  MoveL 1334 to (137.98, -40.97, -45.71) mm, rotated rx -73.13 ry 0 rz 74.07 deg; joints [-2.429, -86.299, 124.187, -182.116, 24.075, 198.51, -176.517]
  MoveL 1335 to (137.95, -41.43, -45.38) mm, rotated rx -73.26 ry 0 rz 73.89 deg; joints [-2.385, -86.31, 124.184, -182.011, 24.075, 198.293, -176.321]
  MoveL 1336 to (137.95, -41.9, -44.95) mm, rotated rx -73.26 ry 0 rz 73.89 deg; joints [-2.363, -86.282, 124.153, -181.958, 24.075, 198.25, -176.318]
  MoveL 1337 to (138.12, -44.92, -41.35) mm, rotated rx -75.02 ry 0 rz 72.24 deg; joints [-1.813, -86.514, 124.201, -180.651, 24.074, 195.429, -174.469]
  MoveL 1338 to (137.32, -48.01, -40.54) mm, rotated rx -75.35 ry 0 rz 70.98 deg; joints [-1.704, -86.538, 124.192, -180.391, 24.074, 194.895, -173.18]
  MoveL 1339 to (137.34, -47.93, -40.55) mm, rotated rx -75.14 ry 0 rz 70.12 deg; joints [-1.748, -86.7, 124.344, -180.494, 24.074, 195.181, -172.312]
  MoveL 1340 to (135.25, -51.11, -43.62) mm, rotated rx -73.93 ry 0 rz 68.65 deg; joints [-2.159, -86.606, 124.375, -181.473, 24.074, 197.191, -170.974]
  MoveL 1341 to (134.45, -52.71, -44.19) mm, rotated rx -73.93 ry 0 rz 68.65 deg; joints [-2.187, -86.465, 124.261, -181.539, 24.075, 197.244, -171.001]
  MoveL 1342 to (134.28, -53.17, -44.17) mm, rotated rx -73.94 ry 0 rz 68.46 deg; joints [-2.183, -86.466, 124.261, -181.53, 24.075, 197.226, -170.805]
  MoveL 1343 to (133.34, -55.46, -44.11) mm, rotated rx -73.97 ry 0 rz 67.44 deg; joints [-2.175, -86.474, 124.266, -181.512, 24.074, 197.187, -169.78]
  MoveL 1344 to (132.43, -57.68, -44.06) mm, rotated rx -73.98 ry 0 rz 66.48 deg; joints [-2.169, -86.476, 124.265, -181.497, 24.074, 197.156, -168.826]
  MoveL 1345 to (132.15, -58.44, -43.91) mm, rotated rx -73.98 ry 0 rz 66.48 deg; joints [-2.161, -86.417, 124.212, -181.478, 24.074, 197.14, -168.832]
  MoveL 1346 to (131.99, -58.95, -43.73) mm, rotated rx -74.06 ry 0 rz 66.28 deg; joints [-2.136, -86.423, 124.21, -181.419, 24.074, 197.018, -168.614]
  MoveL 1347 to (131, -62.6, -41.54) mm, rotated rx -74.84 ry 0 rz 64.98 deg; joints [-1.862, -86.452, 124.16, -180.765, 24.074, 195.708, -167.238]
  MoveL 1348 to (128.38, -67.77, -41.64) mm, rotated rx -74.94 ry 0 rz 62.15 deg; joints [-1.845, -86.56, 124.248, -180.727, 24.074, 195.572, -164.387]
  MoveL 1349 to (145.45, -76.79, -46.84) mm, rotated rx -74.94 ry 0 rz 62.15 deg; joints [-2.108, -87.321, 123.937, -181.362, 24.074, 196.101, -163.319]
  Set speed (1000.0 mm/s)
  MoveL 1350 to (145.71, -79, -42.14) mm, rotated rx -75.13 ry 0 rz 62.13 deg; joints [-1.831, -87.249, 123.803, -180.699, 24.074, 195.37, -163.234]
  Set speed (5.0 mm/s)
  MoveL 1351 to (128.62, -69.96, -37.01) mm, rotated rx -75.13 ry 0 rz 62.13 deg; joints [-1.573, -86.483, 124.11, -180.078, 24.074, 194.858, -164.306]
  Set speed (16.7 mm/s)
  MoveL 1352 to (129.85, -68.52, -35.3) mm, rotated rx -75.8 ry 0 rz 62.86 deg; joints [-1.345, -86.527, 124.09, -179.536, 24.074, 193.748, -164.966]
  MoveL 1353 to (129.85, -68.52, -35.32) mm, rotated rx -76.99 ry 0 rz 63 deg; joints [-1.094, -86.543, 124.043, -178.936, 24.074, 192.069, -165.05]
  MoveL 1354 to (129.74, -69.29, -34.22) mm, rotated rx -77.8 ry 0 rz 62.22 deg; joints [-0.864, -86.677, 124.104, -178.388, 24.074, 190.808, -164.197]
  MoveL 1355 to (129.04, -70.88, -33.63) mm, rotated rx -78.03 ry 0 rz 61.54 deg; joints [-0.785, -86.689, 124.097, -178.199, 24.074, 190.424, -163.504]
  MoveL 1356 to (128.8, -71.45, -33.34) mm, rotated rx -78.08 ry 0 rz 61.44 deg; joints [-0.759, -86.666, 124.071, -178.138, 24.074, 190.321, -163.401]
  MoveL 1357 to (128.09, -73.34, -31.98) mm, rotated rx -78.67 ry 0 rz 60.52 deg; joints [-0.565, -86.719, 124.074, -177.674, 24.074, 189.356, -162.441]
  MoveL 1358 to (127.59, -74.37, -31.59) mm, rotated rx -78.82 ry 0 rz 60.08 deg; joints [-0.513, -86.726, 124.068, -177.549, 24.074, 189.101, -161.985]
  MoveL 1359 to (123.08, -82.67, -28.71) mm, rotated rx -79.95 ry 0 rz 56.4 deg; joints [-0.125, -86.775, 124.03, -176.622, 24.074, 187.214, -158.23]
  MoveL 1360 to (139.48, -93.57, -32.2) mm, rotated rx -79.95 ry 0 rz 56.4 deg; joints [-0.294, -87.571, 123.736, -177.018, 24.074, 187.514, -157.133]
  Set speed (1000.0 mm/s)
  MoveL 1361 to (86.56, -126.27, -76.23) mm, rotated rx -62.7 ry 0 rz 34.53 deg; joints [-6.054, -85.789, 124.002, -190.764, 24.074, 215.943, -137.619]
  Set speed (5.0 mm/s)
  MoveL 1362 to (76.48, -111.63, -67.06) mm, rotated rx -62.7 ry 0 rz 34.53 deg; joints [-5.589, -85.188, 124.406, -189.599, 24.074, 214.927, -138.553]
  Set speed (16.7 mm/s)
  MoveL 1363 to (78.17, -110.46, -67.04) mm, rotated rx -62.7 ry 0 rz 35.27 deg; joints [-5.589, -85.211, 124.425, -189.599, 24.074, 214.927, -139.295]
  MoveL 1364 to (82.31, -108.27, -65.64) mm, rotated rx -63.33 ry 0 rz 37.57 deg; joints [-5.395, -85.243, 124.366, -189.141, 24.074, 213.928, -141.481]
  MoveL 1365 to (83.1, -107.77, -65.47) mm, rotated rx -63.37 ry 0 rz 37.82 deg; joints [-5.379, -85.267, 124.367, -189.118, 24.033, 213.874, -141.742]
  MoveL 1366 to (86.56, -105.46, -64.75) mm, rotated rx -63.68 ry 0 rz 39.58 deg; joints [-5.284, -85.309, 124.362, -188.893, 24.033, 213.389, -143.445]
  MoveL 1367 to (90.08, -104.34, -61.68) mm, rotated rx -65.21 ry 0 rz 41.53 deg; joints [-4.83, -85.421, 124.266, -187.819, 24.033, 211.007, -145.135]
  MoveL 1368 to (92.29, -104.07, -58.82) mm, rotated rx -66.58 ry 0 rz 42.45 deg; joints [-4.417, -85.567, 124.225, -186.84, 24.033, 208.859, -145.827]
  MoveL 1369 to (93.65, -103.42, -57.81) mm, rotated rx -66.58 ry 0 rz 42.45 deg; joints [-4.368, -85.649, 124.225, -186.766, 23.858, 208.808, -145.916]
  MoveL 1370 to (94.29, -102.92, -57.66) mm, rotated rx -66.61 ry 0 rz 42.54 deg; joints [-4.357, -85.68, 124.226, -186.757, 23.785, 208.78, -146.046]
  MoveL 1371 to (95.59, -101.74, -57.6) mm, rotated rx -66.63 ry 0 rz 43.26 deg; joints [-4.348, -85.683, 124.225, -186.737, 23.786, 208.737, -146.762]
  MoveL 1372 to (97.07, -100.77, -56.82) mm, rotated rx -67.03 ry 0 rz 44.34 deg; joints [-4.227, -85.661, 124.161, -186.448, 23.786, 208.107, -147.797]
  MoveL 1373 to (99.36, -99.94, -54.29) mm, rotated rx -68.34 ry 0 rz 45.63 deg; joints [-3.838, -85.738, 124.083, -185.516, 23.786, 206.052, -148.895]
  MoveL 1374 to (99.89, -99.67, -53.81) mm, rotated rx -68.34 ry 0 rz 45.63 deg; joints [-3.814, -85.771, 124.083, -185.472, 23.718, 206.019, -148.928]
  MoveL 1375 to (100.33, -99.39, -53.5) mm, rotated rx -68.42 ry 0 rz 45.75 deg; joints [-3.784, -85.792, 124.084, -185.404, 23.696, 205.89, -149.049]
  MoveL 1376 to (103.28, -97.29, -51.72) mm, rotated rx -69.14 ry 0 rz 47.19 deg; joints [-3.549, -85.876, 124.073, -184.84, 23.696, 204.714, -150.376]
  MoveL 1377 to (103.68, -96.97, -51.52) mm, rotated rx -69.17 ry 0 rz 47.28 deg; joints [-3.533, -85.894, 124.073, -184.805, 23.665, 204.653, -150.482]
  MoveL 1378 to (105.78, -94.99, -50.95) mm, rotated rx -69.35 ry 0 rz 48.27 deg; joints [-3.468, -85.936, 124.074, -184.658, 23.62, 204.355, -151.47]
  MoveL 1379 to (106.4, -94.3, -50.95) mm, rotated rx -69.35 ry 0 rz 48.27 deg; joints [-3.469, -86.006, 124.135, -184.661, 23.62, 204.358, -151.46]
  MoveL 1380 to (106.81, -93.76, -51.06) mm, rotated rx -69.31 ry 0 rz 48.54 deg; joints [-3.485, -86.001, 124.136, -184.698, 23.62, 204.434, -151.739]
  MoveL 1381 to (109.17, -90.01, -52.73) mm, rotated rx -68.69 ry 0 rz 50.1 deg; joints [-3.694, -85.967, 124.18, -185.203, 23.618, 205.459, -153.389]
  MoveL 1382 to (109.1, -90.07, -52.8) mm, rotated rx -68.9 ry 0 rz 51.22 deg; joints [-3.648, -85.766, 123.992, -185.092, 23.618, 205.151, -154.518]
  MoveL 1383 to (110.45, -89.31, -51.3) mm, rotated rx -69.51 ry 0 rz 51.79 deg; joints [-3.451, -85.835, 123.982, -184.615, 23.618, 204.161, -155.002]
  MoveL 1384 to (110.71, -89.18, -50.98) mm, rotated rx -69.68 ry 0 rz 51.94 deg; joints [-3.4, -85.846, 123.974, -184.494, 23.618, 203.894, -155.123]
  MoveL 1385 to (114.23, -86.61, -47.5) mm, rotated rx -70.95 ry 0 rz 53.48 deg; joints [-2.968, -86.008, 123.97, -183.452, 23.618, 201.783, -156.483]
  MoveL 1386 to (115.16, -85.68, -46.95) mm, rotated rx -70.95 ry 0 rz 53.48 deg; joints [-2.942, -86.105, 124.036, -183.392, 23.585, 201.736, -156.483]
  MoveL 1387 to (115.49, -85.28, -46.88) mm, rotated rx -70.98 ry 0 rz 53.69 deg; joints [-2.933, -86.108, 124.036, -183.371, 23.585, 201.692, -156.687]
  MoveL 1388 to (116.72, -83.72, -46.58) mm, rotated rx -71.09 ry 0 rz 54.5 deg; joints [-2.893, -86.116, 124.03, -183.275, 23.585, 201.495, -157.483]
  MoveL 1389 to (117.65, -83.33, -44.95) mm, rotated rx -71.52 ry 0 rz 54.9 deg; joints [-2.724, -86.154, 124.01, -182.866, 23.585, 200.738, -157.816]
  MoveL 1390 to (118.89, -81.86, -44.41) mm, rotated rx -71.96 ry 0 rz 55.31 deg; joints [-2.606, -86.254, 124.06, -182.581, 23.585, 200.066, -158.172]
  MoveL 1391 to (119.23, -81.32, -44.49) mm, rotated rx -71.93 ry 0 rz 55.56 deg; joints [-2.618, -86.251, 124.061, -182.609, 23.585, 200.122, -158.429]
  MoveL 1392 to (122.81, -74.48, -46.64) mm, rotated rx -71.1 ry 0 rz 58.48 deg; joints [-2.897, -86.199, 124.103, -183.283, 23.585, 201.496, -161.446]
  MoveL 1393 to (123.08, -74.04, -46.65) mm, rotated rx -71.07 ry 0 rz 58.84 deg; joints [-2.904, -86.181, 124.102, -183.295, 23.632, 201.537, -161.778]
  MoveL 1394 to (125.13, -70.14, -47.21) mm, rotated rx -70.84 ry 0 rz 60.59 deg; joints [-2.978, -86.159, 124.107, -183.474, 23.632, 201.908, -163.564]
  MoveL 1395 to (125.67, -68.6, -48.04) mm, rotated rx -70.81 ry 0 rz 60.59 deg; joints [-3.029, -86.265, 124.215, -183.596, 23.632, 202.041, -163.568]
  MoveL 1396 to (125.64, -67.91, -49.09) mm, rotated rx -70.78 ry 0 rz 60.59 deg; joints [-3.087, -86.292, 124.256, -183.737, 23.632, 202.179, -163.586]
  MoveL 1397 to (124.81, -67.96, -51.11) mm, rotated rx -70.74 ry 0 rz 60.59 deg; joints [-3.197, -86.235, 124.256, -183.996, 23.676, 202.429, -163.605]
  MoveL 1398 to (123.74, -68.7, -52.68) mm, rotated rx -69.66 ry 0 rz 59.95 deg; joints [-3.498, -86.168, 124.3, -184.721, 23.677, 204.099, -163.092]
  MoveL 1399 to (123.37, -68.58, -53.7) mm, rotated rx -69.24 ry 0 rz 59.92 deg; joints [-3.633, -86.121, 124.306, -185.046, 23.677, 204.775, -163.118]
  MoveL 1400 to (122.17, -69.3, -55.43) mm, rotated rx -67.67 ry 0 rz 59.88 deg; joints [-4.037, -85.916, 124.306, -185.994, 23.78, 207.108, -163.209]
  MoveL 1401 to (122.63, -67.73, -56.41) mm, rotated rx -67.27 ry 0 rz 60.52 deg; joints [-4.165, -85.868, 124.311, -186.3, 23.78, 207.748, -163.921]
  MoveL 1402 to (123.25, -65.21, -58) mm, rotated rx -66.64 ry 0 rz 61.52 deg; joints [-4.371, -85.791, 124.324, -186.793, 23.78, 208.777, -165.028]
  MoveL 1403 to (123.68, -64.08, -58.35) mm, rotated rx -66.37 ry 0 rz 62.29 deg; joints [-4.441, -85.732, 124.324, -186.941, 23.857, 209.16, -165.779]
  MoveL 1404 to (123.84, -63.54, -58.59) mm, rotated rx -66.37 ry 0 rz 62.29 deg; joints [-4.455, -85.77, 124.361, -186.974, 23.857, 209.187, -165.78]
  MoveL 1405 to (124.29, -61.65, -59.63) mm, rotated rx -65.93 ry 0 rz 63.09 deg; joints [-4.593, -85.707, 124.362, -187.304, 23.857, 209.892, -166.655]
  MoveL 1406 to (124.3, -61.62, -59.61) mm, rotated rx -66.05 ry 0 rz 64.34 deg; joints [-4.56, -85.492, 124.167, -187.224, 23.857, 209.703, -167.922]
  MoveL 1407 to (126.02, -59.94, -57.71) mm, rotated rx -66.83 ry 0 rz 65.26 deg; joints [-4.311, -85.596, 124.158, -186.63, 23.857, 208.448, -168.706]
  MoveL 1408 to (128.44, -59.64, -52.46) mm, rotated rx -69.46 ry 0 rz 66.08 deg; joints [-3.521, -85.835, 124.075, -184.743, 23.857, 204.31, -169.145]
  MoveL 1409 to (128.8, -59.51, -51.74) mm, rotated rx -69.54 ry 0 rz 66.1 deg; joints [-3.469, -85.868, 124.085, -184.62, 23.857, 204.13, -169.145]
  MoveL 1410 to (129.78, -58.91, -49.96) mm, rotated rx -70.26 ry 0 rz 66.48 deg; joints [-3.233, -85.946, 124.072, -184.057, 23.855, 202.958, -169.423]
  MoveL 1411 to (130.23, -58.65, -49.07) mm, rotated rx -70.48 ry 0 rz 66.57 deg; joints [-3.143, -85.991, 124.081, -183.841, 23.855, 202.559, -169.462]
  MoveL 1412 to (132.89, -56.13, -44.69) mm, rotated rx -72.23 ry 0 rz 67.91 deg; joints [-2.565, -86.163, 124.047, -182.456, 23.855, 199.694, -170.572]
  MoveL 1413 to (133.87, -54.54, -43.72) mm, rotated rx -72.23 ry 0 rz 67.91 deg; joints [-2.517, -86.301, 124.138, -182.348, 23.806, 199.607, -170.572]
  MoveL 1414 to (134.4, -52.63, -44.42) mm, rotated rx -72.23 ry 0 rz 67.91 deg; joints [-2.555, -86.439, 124.266, -182.438, 23.802, 199.68, -170.568]
  MoveL 1415 to (134.45, -52.04, -44.98) mm, rotated rx -72.01 ry 0 rz 68.13 deg; joints [-2.628, -86.418, 124.271, -182.615, 23.802, 200.044, -170.823]
  MoveL 1416 to (134.35, -51.3, -46.09) mm, rotated rx -72.01 ry 0 rz 68.13 deg; joints [-2.685, -86.451, 124.317, -182.75, 23.802, 200.154, -170.838]
  MoveL 1417 to (132.92, -49.01, -52.29) mm, rotated rx -68.94 ry 0 rz 69.21 deg; joints [-3.624, -86.082, 124.317, -184.994, 23.838, 205.029, -172.299]
  MoveL 1418 to (133.31, -45.82, -54.18) mm, rotated rx -68.18 ry 0 rz 70.48 deg; joints [-3.873, -85.993, 124.328, -185.589, 23.838, 206.272, -173.685]
  MoveL 1419 to (133.02, -44.52, -55.95) mm, rotated rx -68.18 ry 0 rz 70.48 deg; joints [-3.963, -86.046, 124.406, -185.806, 23.838, 206.446, -173.717]
  MoveL 1420 to (132.73, -44.42, -56.71) mm, rotated rx -68.1 ry 0 rz 70.49 deg; joints [-4.017, -86.023, 124.406, -185.936, 23.838, 206.629, -173.751]
  MoveL 1421 to (132.12, -44.47, -58.08) mm, rotated rx -67.54 ry 0 rz 70.38 deg; joints [-4.198, -85.953, 124.414, -186.368, 23.838, 207.536, -173.74]
  MoveL 1422 to (131.58, -43.17, -60.26) mm, rotated rx -66.1 ry 0 rz 70.89 deg; joints [-4.592, -85.779, 124.417, -187.308, 23.838, 209.722, -174.459]
  MoveL 1423 to (131.38, -42.9, -60.88) mm, rotated rx -66.1 ry 0 rz 70.89 deg; joints [-4.624, -85.78, 124.431, -187.384, 23.838, 209.782, -174.474]
  MoveL 1424 to (131.19, -42.76, -61.38) mm, rotated rx -65.89 ry 0 rz 70.92 deg; joints [-4.69, -85.752, 124.433, -187.542, 23.838, 210.117, -174.541]
  MoveL 1425 to (130.01, -41.88, -64.4) mm, rotated rx -64.63 ry 0 rz 71.11 deg; joints [-5.089, -85.574, 124.446, -188.493, 23.838, 212.139, -174.964]
  MoveL 1426 to (130.03, -41.89, -64.35) mm, rotated rx -63.97 ry 0 rz 71.59 deg; joints [-5.213, -85.465, 124.446, -188.743, 23.975, 212.984, -175.43]
  MoveL 1427 to (130.19, -37.44, -66.76) mm, rotated rx -62.96 ry 0 rz 73.39 deg; joints [-5.527, -85.314, 124.456, -189.488, 23.975, 214.583, -177.435]
  MoveL 1428 to (129.62, -36.05, -68.6) mm, rotated rx -62.96 ry 0 rz 73.39 deg; joints [-5.622, -85.357, 124.534, -189.714, 23.975, 214.762, -177.483]
  MoveL 1429 to (129.03, -35.2, -70.14) mm, rotated rx -62.01 ry 0 rz 73.73 deg; joints [-5.88, -85.215, 124.534, -190.323, 23.978, 216.195, -177.992]
  MoveL 1430 to (128.75, -34.95, -70.79) mm, rotated rx -61.95 ry 0 rz 73.75 deg; joints [-5.923, -85.204, 124.543, -190.423, 23.978, 216.325, -178.035]
  MoveL 1431 to (128.62, -34.84, -71.06) mm, rotated rx -61.16 ry 0 rz 74.22 deg; joints [-6.085, -85.07, 124.543, -190.76, 24.099, 217.374, -178.54]
  MoveL 1432 to (128.52, -33.37, -71.94) mm, rotated rx -60.78 ry 0 rz 74.81 deg; joints [-6.199, -85.009, 124.547, -191.029, 24.099, 217.961, -179.22]
  MoveL 1433 to (128.3, -32.51, -72.73) mm, rotated rx -60.78 ry 0 rz 74.81 deg; joints [-6.241, -85.045, 124.597, -191.128, 24.099, 218.039, -179.24]
  MoveL 1434 to (128.05, -32.17, -73.32) mm, rotated rx -60.73 ry 0 rz 74.84 deg; joints [-6.28, -85.039, 124.611, -191.219, 24.099, 218.159, -179.294]
  MoveL 1435 to (127.47, -31.67, -74.53) mm, rotated rx -60.2 ry 0 rz 74.99 deg; joints [-6.438, -84.951, 124.616, -191.591, 24.099, 218.974, -179.554]
  MoveL 1436 to (126.85, -29.7, -76.38) mm, rotated rx -59.02 ry 0 rz 75.96 deg; joints [-6.771, -84.988, 125.113, -191.94, 25.126, 220.344, -180]
  MoveL 1437 to (126.72, -29.34, -76.74) mm, rotated rx -58.91 ry 0 rz 76.06 deg; joints [-6.814, -85.013, 125.204, -191.969, 25.294, 220.465, -180]
  MoveL 1438 to (125.84, -27.3, -78.9) mm, rotated rx -57.96 ry 0 rz 76.84 deg; joints [-7.131, -85.152, 125.88, -192.137, 26.641, 221.44, -180]
  MoveL 1439 to (125.36, -26.75, -79.85) mm, rotated rx -57.96 ry 0 rz 76.84 deg; joints [-7.181, -85.165, 125.931, -192.227, 26.686, 221.505, -180]
  MoveL 1440 to (124.53, -26.64, -81.17) mm, rotated rx -57.8 ry 0 rz 76.87 deg; joints [-7.277, -85.126, 125.99, -192.382, 26.821, 221.763, -180]
  MoveL 1441 to (122.66, -27.32, -83.76) mm, rotated rx -56.63 ry 0 rz 76.37 deg; joints [-7.618, -84.902, 125.994, -193.109, 26.821, 223.479, -179.787]
  MoveL 1442 to (120.31, -27.21, -87.13) mm, rotated rx -54.87 ry 0 rz 76.1 deg; joints [-8.096, -84.582, 126.011, -194.127, 26.821, 225.985, -179.937]
  MoveL 1443 to (119.84, -27.31, -87.74) mm, rotated rx -54.87 ry 0 rz 76.1 deg; joints [-8.125, -84.551, 126.011, -194.178, 26.848, 226.019, -179.947]
  MoveL 1444 to (119.51, -27.47, -88.15) mm, rotated rx -54.68 ry 0 rz 75.99 deg; joints [-8.179, -84.513, 126.012, -194.292, 26.848, 226.294, -179.886]
  MoveL 1445 to (115.59, -30.1, -92.42) mm, rotated rx -52.79 ry 0 rz 74.41 deg; joints [-8.711, -84.104, 126.015, -195.418, 26.848, 228.993, -178.81]
  MoveL 1446 to (115.26, -30.28, -92.76) mm, rotated rx -52.59 ry 0 rz 74.25 deg; joints [-8.762, -84.07, 126.021, -195.526, 26.848, 229.272, -178.705]
  MoveL 1447 to (111.45, -33.08, -96.4) mm, rotated rx -50.93 ry 0 rz 72.51 deg; joints [-9.215, -83.699, 126.028, -196.481, 26.848, 231.613, -177.43]
  MoveL 1448 to (110.88, -33.62, -96.87) mm, rotated rx -50.85 ry 0 rz 72.38 deg; joints [-9.25, -83.65, 126.028, -196.526, 26.9, 231.715, -177.302]
  MoveL 1449 to (109.03, -35.76, -98.19) mm, rotated rx -50.24 ry 0 rz 71.16 deg; joints [-9.414, -83.504, 126.028, -196.869, 26.901, 232.572, -176.255]
  MoveL 1450 to (105.97, -37.85, -100.72) mm, rotated rx -48.8 ry 0 rz 69.4 deg; joints [-9.771, -83.244, 126.083, -197.617, 26.901, 234.531, -174.884]
  MoveL 1451 to (105.56, -38.13, -101.04) mm, rotated rx -48.65 ry 0 rz 69.21 deg; joints [-9.81, -83.208, 126.083, -197.698, 26.901, 234.736, -174.743]
  MoveL 1452 to (102.4, -40.39, -103.39) mm, rotated rx -47.47 ry 0 rz 67.57 deg; joints [-10.109, -82.943, 126.104, -198.318, 26.901, 236.342, -173.448]
  MoveL 1453 to (101.99, -40.57, -103.73) mm, rotated rx -47.27 ry 0 rz 67.37 deg; joints [-10.157, -82.905, 126.112, -198.417, 26.901, 236.61, -173.305]
  MoveL 1454 to (97.91, -42.95, -106.66) mm, rotated rx -45.71 ry 0 rz 65.33 deg; joints [-10.536, -82.565, 126.153, -199.2, 26.901, 238.696, -171.734]
  MoveL 1455 to (96.76, -44.15, -107.22) mm, rotated rx -45.71 ry 0 rz 65.33 deg; joints [-10.552, -82.429, 126.069, -199.214, 26.926, 238.696, -171.762]
  MoveL 1456 to (95.06, -46.9, -107.57) mm, rotated rx -45.52 ry 0 rz 63.53 deg; joints [-10.599, -82.396, 126.083, -199.311, 26.926, 238.956, -170.017]
  MoveL 1457 to (92.2, -49.19, -109.03) mm, rotated rx -44.59 ry 0 rz 61.21 deg; joints [-10.814, -82.269, 126.168, -199.753, 26.926, 240.175, -167.952]
  MoveL 1458 to (91.24, -50.42, -109.28) mm, rotated rx -44.59 ry 0 rz 61.21 deg; joints [-10.814, -82.145, 126.073, -199.749, 26.927, 240.167, -167.981]
  MoveL 1459 to (90.83, -51.64, -109.04) mm, rotated rx -44.6 ry 0 rz 61.05 deg; joints [-10.793, -82.085, 126.01, -199.705, 26.927, 240.124, -167.816]
  MoveL 1460 to (90.6, -53.29, -108.43) mm, rotated rx -44.94 ry 0 rz 60.2 deg; joints [-10.715, -82.159, 126, -199.544, 26.928, 239.685, -166.862]
  MoveL 1461 to (90.59, -53.38, -108.39) mm, rotated rx -45.04 ry 0 rz 59.12 deg; joints [-10.712, -82.315, 126.115, -199.544, 26.925, 239.586, -165.746]
  MoveL 1462 to (89.12, -54.97, -108.83) mm, rotated rx -44.81 ry 0 rz 57.95 deg; joints [-10.768, -82.263, 126.123, -199.658, 26.925, 239.897, -164.653]
  MoveL 1463 to (88.6, -55.68, -108.89) mm, rotated rx -44.81 ry 0 rz 57.95 deg; joints [-10.764, -82.196, 126.069, -199.649, 26.925, 239.888, -164.665]
  MoveL 1464 to (88.21, -56.59, -108.74) mm, rotated rx -44.81 ry 0 rz 57.86 deg; joints [-10.749, -82.144, 126.017, -199.617, 26.925, 239.86, -164.569]
  MoveL 1465 to (87.77, -58.17, -108.26) mm, rotated rx -45.07 ry 0 rz 57.01 deg; joints [-10.688, -82.202, 126.008, -199.491, 26.925, 239.515, -163.635]
  MoveL 1466 to (87.47, -59.22, -107.93) mm, rotated rx -45.14 ry 0 rz 56.72 deg; joints [-10.658, -82.188, 125.973, -199.429, 26.925, 239.406, -163.314]
  MoveL 1467 to (87.01, -63.11, -106.08) mm, rotated rx -46.14 ry 0 rz 54.84 deg; joints [-10.419, -82.41, 125.945, -198.939, 26.925, 238.081, -161.137]
  MoveL 1468 to (87.5, -64.69, -104.72) mm, rotated rx -46.14 ry 0 rz 54.84 deg; joints [-10.346, -82.395, 125.874, -198.786, 26.925, 237.975, -161.064]
  MoveL 1469 to (88.16, -65.07, -103.92) mm, rotated rx -46.27 ry 0 rz 54.83 deg; joints [-10.288, -82.454, 125.873, -198.668, 26.925, 237.766, -160.984]
  MoveL 1470 to (89.29, -65.35, -102.77) mm, rotated rx -46.86 ry 0 rz 55.05 deg; joints [-10.142, -82.585, 125.859, -198.365, 26.925, 236.966, -161.024]
  MoveL 1471 to (89.25, -65.37, -102.8) mm, rotated rx -47.65 ry 0 rz 54.83 deg; joints [-10.024, -82.715, 125.859, -198.136, 26.897, 236.026, -160.675]
  MoveL 1472 to (89.38, -66.4, -102.03) mm, rotated rx -48.05 ry 0 rz 54.43 deg; joints [-9.923, -82.803, 125.85, -197.929, 26.897, 235.481, -160.163]
  MoveL 1473 to (90.2, -67.77, -100.38) mm, rotated rx -49.14 ry 0 rz 52.4 deg; joints [-9.682, -83.185, 125.85, -197.66, 26.483, 234.283, -158.129]
  MoveL 1474 to (88.7, -68.61, -101.15) mm, rotated rx -48.75 ry 0 rz 51.59 deg; joints [-9.782, -83.102, 125.858, -197.87, 26.483, 234.818, -157.429]
  MoveL 1475 to (87.69, -69.33, -101.54) mm, rotated rx -48.76 ry 0 rz 51.56 deg; joints [-9.79, -83.004, 125.788, -197.886, 26.483, 234.814, -157.426]
  MoveL 1476 to (86.89, -70.89, -101.15) mm, rotated rx -48.78 ry 0 rz 51.52 deg; joints [-9.757, -82.902, 125.683, -197.813, 26.483, 234.742, -157.372]
  MoveL 1477 to (87.23, -72.68, -99.58) mm, rotated rx -48.8 ry 0 rz 51.46 deg; joints [-9.67, -82.89, 125.608, -197.627, 26.483, 234.587, -157.233]
  MoveL 1478 to (88.09, -73.52, -98.19) mm, rotated rx -49.5 ry 0 rz 51.4 deg; joints [-9.492, -83.038, 125.595, -197.251, 26.483, 233.627, -156.977]
  MoveL 1479 to (88.4, -75.8, -96.15) mm, rotated rx -51.34 ry 0 rz 49.82 deg; joints [-9.098, -83.448, 125.595, -196.505, 26.319, 231.279, -155.075]
  MoveL 1480 to (86.63, -79.11, -95.09) mm, rotated rx -51.86 ry 0 rz 48.02 deg; joints [-8.961, -83.557, 125.587, -196.21, 26.319, 230.548, -153.136]
  MoveL 1481 to (86.26, -79.54, -95.08) mm, rotated rx -51.93 ry 0 rz 47.44 deg; joints [-8.953, -83.606, 125.612, -196.211, 26.287, 230.491, -152.557]
  MoveL 1482 to (79.34, -84.7, -96.64) mm, rotated rx -51.14 ry 0 rz 42.85 deg; joints [-9.164, -83.502, 125.673, -196.663, 26.287, 231.6, -148.18]
  MoveL 1483 to (78.82, -85.12, -96.69) mm, rotated rx -51.14 ry 0 rz 42.72 deg; joints [-9.165, -83.47, 125.649, -196.663, 26.29, 231.605, -148.057]
  MoveL 1484 to (77.12, -86.67, -96.68) mm, rotated rx -51.14 ry 0 rz 41.67 deg; joints [-9.162, -83.459, 125.639, -196.658, 26.29, 231.595, -147.006]
  MoveL 1485 to (76.85, -86.83, -96.76) mm, rotated rx -51.08 ry 0 rz 41.23 deg; joints [-9.18, -83.491, 125.677, -196.696, 26.29, 231.685, -146.572]
  MoveL 1486 to (70.66, -88.85, -99.6) mm, rotated rx -49.55 ry 0 rz 37.84 deg; joints [-9.572, -83.23, 125.748, -197.534, 26.29, 233.813, -143.599]
  MoveL 1487 to (69.62, -89.36, -99.87) mm, rotated rx -49.55 ry 0 rz 37.84 deg; joints [-9.577, -83.137, 125.681, -197.54, 26.297, 233.813, -143.618]
  MoveL 1488 to (68.94, -89.84, -99.91) mm, rotated rx -49.53 ry 0 rz 37.42 deg; joints [-9.583, -83.132, 125.681, -197.551, 26.297, 233.841, -143.203]
  MoveL 1489 to (62.76, -94.08, -100.08) mm, rotated rx -49.44 ry 0 rz 33.67 deg; joints [-9.604, -83.109, 125.681, -197.592, 26.305, 233.954, -139.473]
  MoveL 1490 to (62.53, -94.11, -100.2) mm, rotated rx -49.32 ry 0 rz 33.16 deg; joints [-9.634, -83.147, 125.733, -197.657, 26.305, 234.119, -138.984]
  MoveL 1491 to (54.8, -96.96, -101.99) mm, rotated rx -48.43 ry 0 rz 29.11 deg; joints [-9.862, -82.943, 125.742, -198.14, 26.305, 235.349, -135.194]
  MoveL 1492 to (52.96, -98.33, -101.65) mm, rotated rx -48.43 ry 0 rz 29.11 deg; joints [-9.829, -82.789, 125.597, -198.066, 26.305, 235.292, -135.195]
  MoveL 1493 to (52.64, -98.87, -101.3) mm, rotated rx -48.51 ry 0 rz 28.97 deg; joints [-9.797, -82.795, 125.578, -197.997, 26.305, 235.158, -135.022]
  MoveL 1494 to (51.49, -101.18, -99.59) mm, rotated rx -49.39 ry 0 rz 27.89 deg; joints [-9.576, -82.982, 125.56, -197.529, 26.305, 233.959, -133.691]
  MoveL 1495 to (51.53, -102.66, -98.05) mm, rotated rx -49.39 ry 0 rz 27.89 deg; joints [-9.496, -82.995, 125.513, -197.359, 26.305, 233.838, -133.614]
  MoveL 1496 to (52.62, -103.3, -96.79) mm, rotated rx -49.5 ry 0 rz 27.91 deg; joints [-9.418, -83.093, 125.513, -197.233, 26.234, 233.643, -133.594]
  MoveL 1497 to (54.87, -103.58, -95.22) mm, rotated rx -50.27 ry 0 rz 28.82 deg; joints [-9.22, -83.255, 125.5, -196.808, 26.234, 232.578, -134.283]
  MoveL 1498 to (56.61, -104.63, -93.02) mm, rotated rx -52.15 ry 0 rz 29.6 deg; joints [-8.8, -83.536, 125.438, -195.907, 26.234, 230.054, -134.637]
  MoveL 1499 to (56.93, -106.13, -91.13) mm, rotated rx -53.06 ry 0 rz 29.38 deg; joints [-8.554, -83.722, 125.427, -195.378, 26.234, 228.76, -134.174]
  MoveL 1500 to (57.12, -106.52, -90.54) mm, rotated rx -53.06 ry 0 rz 29.38 deg; joints [-8.526, -83.741, 125.424, -195.316, 26.234, 228.715, -134.147]
  MoveL 1501 to (57.34, -106.77, -90.11) mm, rotated rx -53.16 ry 0 rz 29.39 deg; joints [-8.487, -83.772, 125.424, -195.234, 26.232, 228.551, -134.124]
  MoveL 1502 to (58.34, -107.62, -88.43) mm, rotated rx -53.95 ry 0 rz 29.6 deg; joints [-8.271, -83.931, 125.416, -194.768, 26.232, 227.425, -134.129]
  MoveL 1503 to (58.38, -109.47, -86.11) mm, rotated rx -55.51 ry 0 rz 29.17 deg; joints [-7.888, -84.206, 125.408, -193.939, 26.231, 225.258, -133.346]
  MoveL 1504 to (58.45, -109.83, -85.61) mm, rotated rx -55.56 ry 0 rz 29.17 deg; joints [-7.853, -84.223, 125.401, -193.863, 26.231, 225.146, -133.309]
  MoveL 1505 to (58.95, -110.73, -84.09) mm, rotated rx -56.15 ry 0 rz 29.17 deg; joints [-7.676, -84.343, 125.395, -193.478, 26.231, 224.277, -133.16]
  MoveL 1506 to (59.03, -111.65, -82.81) mm, rotated rx -56.95 ry 0 rz 28.97 deg; joints [-7.471, -84.484, 125.394, -193.034, 26.231, 223.148, -132.782]
  MoveL 1507 to (59.46, -112.26, -81.67) mm, rotated rx -56.95 ry 0 rz 28.97 deg; joints [-7.415, -84.525, 125.394, -192.916, 26.223, 223.06, -132.74]
  MoveL 1508 to (60.36, -112.5, -80.66) mm, rotated rx -57.04 ry 0 rz 29.01 deg; joints [-7.35, -84.596, 125.394, -192.804, 26.149, 222.887, -132.774]
  MoveL 1509 to (61.18, -112.49, -80.06) mm, rotated rx -57.31 ry 0 rz 29.33 deg; joints [-7.271, -84.646, 125.393, -192.633, 26.149, 222.489, -133.03]
  MoveL 1510 to (61.19, -112.52, -80) mm, rotated rx -58.25 ry 0 rz 29.62 deg; joints [-7.096, -84.707, 125.348, -192.251, 26.149, 221.269, -133.183]
  MoveL 1511 to (61.24, -113.39, -78.74) mm, rotated rx -58.81 ry 0 rz 29.45 deg; joints [-6.931, -84.81, 125.345, -191.89, 26.149, 220.434, -132.879]
  MoveL 1512 to (61.37, -113.79, -78.05) mm, rotated rx -58.81 ry 0 rz 29.45 deg; joints [-6.897, -84.825, 125.34, -191.815, 26.149, 220.377, -132.853]
  MoveL 1513 to (61.99, -114.24, -76.9) mm, rotated rx -58.93 ry 0 rz 29.46 deg; joints [-6.819, -84.887, 125.34, -191.658, 26.113, 220.141, -132.826]
  MoveL 1514 to (64.03, -114.71, -74.5) mm, rotated rx -59.98 ry 0 rz 30.12 deg; joints [-6.505, -85.074, 125.336, -190.972, 26.113, 218.569, -133.257]
  MoveL 1515 to (64.8, -115.27, -72.94) mm, rotated rx -60.89 ry 0 rz 30.39 deg; joints [-6.258, -85.197, 125.317, -190.429, 26.113, 217.25, -133.349]
  MoveL 1516 to (65.55, -115.43, -72.01) mm, rotated rx -60.89 ry 0 rz 30.39 deg; joints [-6.213, -85.248, 125.317, -190.353, 26.041, 217.198, -133.365]
  MoveL 1517 to (66.58, -115.27, -71.33) mm, rotated rx -60.95 ry 0 rz 30.46 deg; joints [-6.167, -85.309, 125.317, -190.289, 25.938, 217.089, -133.471]
  MoveL 1518 to (69.19, -114.39, -70.25) mm, rotated rx -61.42 ry 0 rz 31.61 deg; joints [-6.026, -85.387, 125.315, -189.977, 25.938, 216.385, -134.523]
  MoveL 1519 to (69.84, -114.17, -69.96) mm, rotated rx -61.55 ry 0 rz 31.92 deg; joints [-5.987, -85.405, 125.312, -189.891, 25.938, 216.19, -134.802]
  MoveL 1520 to (75.72, -112.02, -67.28) mm, rotated rx -62.7 ry 0 rz 34.53 deg; joints [-5.634, -85.589, 125.305, -189.109, 25.938, 214.438, -137.175]
  MoveL 1521 to (85.79, -126.66, -76.45) mm, rotated rx -62.7 ry 0 rz 34.53 deg; joints [-6.105, -86.221, 124.93, -190.209, 25.938, 215.391, -136.236]
  Set speed (1000.0 mm/s)
  MoveL 1522 to (70.78, -152.61, -30.8) mm, rotated rx -80.27 ry 0 rz 24.34 deg; joints [-0.137, -88.324, 124.915, -176.855, 25.938, 187.083, -123.644]
  Set speed (5.0 mm/s)
  MoveL 1523 to (62.66, -134.65, -27.42) mm, rotated rx -80.27 ry 0 rz 24.34 deg; joints [0.028, -87.493, 125.176, -176.494, 25.938, 186.819, -124.744]
  Set speed (16.7 mm/s)
  MoveL 1524 to (60.97, -135.12, -28.83) mm, rotated rx -79.73 ry 0 rz 23.67 deg; joints [-0.163, -87.473, 125.197, -176.922, 25.938, 187.712, -124.105]
  MoveL 1525 to (60.92, -135.13, -28.89) mm, rotated rx -79.14 ry 0 rz 23.32 deg; joints [-0.294, -87.487, 125.197, -177.203, 25.806, 188.523, -123.866]
  MoveL 1526 to (60.25, -134.81, -31.58) mm, rotated rx -78.09 ry 0 rz 23.12 deg; joints [-0.658, -87.44, 125.233, -178.023, 25.806, 190.233, -123.744]
  MoveL 1527 to (67.93, -152.81, -35.71) mm, rotated rx -78.09 ry 0 rz 23.12 deg; joints [-0.865, -88.258, 124.966, -178.484, 25.807, 190.593, -122.653]
  Set speed (1000.0 mm/s)
  MoveL 1528 to (62.13, -154.29, -39.73) mm, rotated rx -77.4 ry 0 rz 21.89 deg; joints [-1.221, -88.026, 124.84, -179.288, 25.807, 191.94, -121.517]
  Set speed (5.0 mm/s)
  MoveL 1529 to (54.86, -136.18, -35.37) mm, rotated rx -77.4 ry 0 rz 21.89 deg; joints [-1.002, -87.213, 125.112, -178.795, 25.807, 191.548, -122.604]
  Set speed (16.7 mm/s)
  MoveL 1530 to (54.31, -136.4, -35.4) mm, rotated rx -77.39 ry 0 rz 21.66 deg; joints [-1.006, -87.213, 125.112, -178.805, 25.807, 191.568, -122.376]
  MoveL 1531 to (53.04, -136.99, -35.06) mm, rotated rx -77.39 ry 0 rz 21.66 deg; joints [-0.99, -87.111, 125.018, -178.768, 25.807, 191.538, -122.385]
  MoveL 1532 to (52.22, -137.43, -34.53) mm, rotated rx -77.6 ry 0 rz 21.3 deg; joints [-0.918, -87.122, 125.012, -178.607, 25.807, 191.2, -122.007]
  MoveL 1533 to (45.37, -141.15, -28.72) mm, rotated rx -79.79 ry 0 rz 18.41 deg; joints [-0.149, -87.206, 124.919, -176.877, 25.807, 187.611, -118.965]
  MoveL 1534 to (45.01, -141.33, -28.39) mm, rotated rx -79.89 ry 0 rz 18.29 deg; joints [-0.111, -87.203, 124.908, -176.792, 25.807, 187.444, -118.843]
  MoveL 1535 to (42.69, -142.49, -26.11) mm, rotated rx -80.75 ry 0 rz 17.32 deg; joints [0.192, -87.227, 124.871, -176.109, 25.808, 186.029, -117.828]
  MoveL 1536 to (42.3, -142.7, -25.61) mm, rotated rx -80.75 ry 0 rz 17.32 deg; joints [0.217, -87.196, 124.84, -176.053, 25.808, 185.984, -117.828]
  MoveL 1537 to (42.08, -142.83, -25.21) mm, rotated rx -80.9 ry 0 rz 17.23 deg; joints [0.271, -87.2, 124.833, -175.932, 25.808, 185.732, -117.721]
  MoveL 1538 to (40.3, -143.93, -21.61) mm, rotated rx -82.23 ry 0 rz 16.48 deg; joints [0.744, -87.222, 124.769, -174.866, 25.808, 183.535, -116.919]
  MoveL 1539 to (37.44, -145.06, -19.09) mm, rotated rx -83.46 ry 0 rz 15.09 deg; joints [1.142, -87.275, 124.753, -173.966, 25.808, 181.575, -115.492]
  MoveL 1540 to (37.01, -145.23, -18.58) mm, rotated rx -83.46 ry 0 rz 15.09 deg; joints [1.167, -87.259, 124.753, -173.921, 25.871, 181.541, -115.448]
  MoveL 1541 to (36.66, -145.4, -17.96) mm, rotated rx -83.58 ry 0 rz 15.01 deg; joints [1.224, -87.256, 124.752, -173.801, 25.907, 181.329, -115.341]
  MoveL 1542 to (35.62, -145.92, -15.58) mm, rotated rx -84.48 ry 0 rz 14.58 deg; joints [1.543, -87.256, 124.709, -173.083, 25.913, 179.838, -114.886]
  MoveL 1543 to (33.5, -146.58, -14.11) mm, rotated rx -85.43 ry 0 rz 13.4 deg; joints [1.829, -87.315, 124.723, -172.439, 25.913, 178.364, -113.689]
  MoveL 1544 to (33.07, -146.71, -13.74) mm, rotated rx -85.49 ry 0 rz 13.33 deg; joints [1.859, -87.305, 124.723, -172.381, 25.957, 178.264, -113.596]
  MoveL 1545 to (31.61, -147.19, -11.93) mm, rotated rx -86.07 ry 0 rz 12.86 deg; joints [2.08, -87.302, 124.723, -171.91, 26.055, 177.302, -113.045]
  MoveL 1546 to (31.23, -147.3, -11.66) mm, rotated rx -86.3 ry 0 rz 12.58 deg; joints [2.145, -87.323, 124.734, -171.764, 26.055, 176.953, -112.766]
  MoveL 1547 to (25.25, -148.78, -5.86) mm, rotated rx -88.47 ry 0 rz 10.29 deg; joints [2.919, -87.323, 124.734, -170.109, 26.32, 173.458, -110.303]
  MoveL 1548 to (24.36, -148.99, -4.06) mm, rotated rx -88.49 ry 0 rz 10.32 deg; joints [3.013, -87.281, 124.734, -169.949, 26.472, 173.314, -110.236]
  MoveL 1549 to (24.52, -148.98, -3.15) mm, rotated rx -88.5 ry 0 rz 10.33 deg; joints [3.062, -87.284, 124.733, -169.84, 26.472, 173.216, -110.252]
  MoveL 1550 to (25.82, -148.79, -1.69) mm, rotated rx -88.52 ry 0 rz 10.36 deg; joints [3.146, -87.366, 124.799, -169.654, 26.472, 173.044, -110.278]
  MoveL 1551 to (27.78, -148.44, -1.42) mm, rotated rx -88.54 ry 0 rz 10.39 deg; joints [3.172, -87.506, 124.921, -169.594, 26.473, 172.974, -110.293]
  MoveL 1552 to (31.01, -147.79, -2.17) mm, rotated rx -88.25 ry 0 rz 11.64 deg; joints [3.07, -87.509, 124.921, -169.809, 26.437, 173.432, -111.559]
  MoveL 1553 to (33.69, -147.2, -2.25) mm, rotated rx -88.2 ry 0 rz 12.86 deg; joints [3.053, -87.476, 124.893, -169.848, 26.437, 173.517, -112.781]
  MoveL 1554 to (34.44, -147.02, -2.4) mm, rotated rx -88.2 ry 0 rz 12.86 deg; joints [3.048, -87.527, 124.931, -169.85, 26.411, 173.517, -112.793]
  MoveL 1555 to (34.9, -146.91, -2.57) mm, rotated rx -88.13 ry 0 rz 13.04 deg; joints [3.025, -87.527, 124.931, -169.9, 26.403, 173.622, -112.977]
  MoveL 1556 to (35.62, -146.73, -3) mm, rotated rx -88.13 ry 0 rz 13.04 deg; joints [3.004, -87.558, 124.931, -169.914, 26.306, 173.628, -113.041]
  MoveL 1557 to (39.46, -145.64, -6.33) mm, rotated rx -86.87 ry 0 rz 14.55 deg; joints [2.553, -87.562, 124.931, -170.875, 26.155, 175.665, -114.642]
  MoveL 1558 to (41.08, -145.14, -7.17) mm, rotated rx -86.44 ry 0 rz 15.37 deg; joints [2.415, -87.538, 124.925, -171.186, 26.155, 176.349, -115.459]
  MoveL 1559 to (46.37, -164.39, -8.41) mm, rotated rx -86.44 ry 0 rz 15.37 deg; joints [2.371, -88.383, 124.664, -171.256, 26.155, 176.329, -114.351]
  Set speed (1000.0 mm/s)
  MoveL 1560 to (62.65, -157.67, -21.45) mm, rotated rx -82.12 ry 0 rz 21.17 deg; joints [0.748, -88.384, 124.82, -174.865, 25.963, 183.605, -120.347]
  Set speed (5.0 mm/s)
  MoveL 1561 to (55.49, -139.2, -18.7) mm, rotated rx -82.12 ry 0 rz 21.17 deg; joints [0.876, -87.544, 125.077, -174.593, 25.963, 183.429, -121.453]
  Set speed (16.7 mm/s)
  MoveL 1562 to (56.32, -138.78, -19.37) mm, rotated rx -81.86 ry 0 rz 21.52 deg; joints [0.787, -87.541, 125.089, -174.795, 25.963, 183.847, -121.813]
  MoveL 1563 to (56.8, -138.51, -19.87) mm, rotated rx -81.77 ry 0 rz 21.62 deg; joints [0.741, -87.548, 125.09, -174.89, 25.915, 184.016, -121.943]
  MoveL 1564 to (57.53, -138.1, -20.62) mm, rotated rx -81.45 ry 0 rz 21.97 deg; joints [0.632, -87.536, 125.097, -175.133, 25.915, 184.535, -122.313]
  MoveL 1565 to (57.56, -138.08, -20.68) mm, rotated rx -81.26 ry 0 rz 23.02 deg; joints [0.583, -87.332, 124.925, -175.245, 25.915, 184.814, -123.385]
  MoveL 1566 to (58.55, -137.73, -20.22) mm, rotated rx -81.44 ry 0 rz 23.42 deg; joints [0.645, -87.335, 124.917, -175.106, 25.915, 184.526, -123.78]
  MoveL 1567 to (60.3, -136.98, -20.17) mm, rotated rx -81.44 ry 0 rz 23.42 deg; joints [0.651, -87.477, 125.042, -175.092, 25.915, 184.513, -123.763]
  MoveL 1568 to (61.39, -136.38, -20.98) mm, rotated rx -81.41 ry 0 rz 23.5 deg; joints [0.604, -87.514, 125.042, -175.175, 25.778, 184.606, -123.939]
  MoveL 1569 to (63.29, -135.06, -23.68) mm, rotated rx -80.37 ry 0 rz 24.37 deg; joints [0.24, -87.491, 125.087, -175.997, 25.778, 186.311, -124.855]
  MoveL 1570 to (71.42, -153.02, -27.03) mm, rotated rx -80.37 ry 0 rz 24.37 deg; joints [0.078, -88.322, 124.825, -176.352, 25.778, 186.567, -123.755]
  Set speed (1000.0 mm/s)
  MoveL 1571 to (90.43, -139.29, -40.79) mm, rotated rx -75.42 ry 0 rz 32.69 deg; joints [-1.704, -87.978, 124.905, -180.376, 25.778, 194.813, -132.463]
  Set speed (5.0 mm/s)
  MoveL 1572 to (79.98, -123, -35.75) mm, rotated rx -75.42 ry 0 rz 32.69 deg; joints [-1.448, -87.179, 125.182, -179.797, 25.778, 194.342, -133.538]
  Set speed (16.7 mm/s)
  MoveL 1573 to (83.77, -119.93, -37.51) mm, rotated rx -74.73 ry 0 rz 34.59 deg; joints [-1.684, -87.13, 125.199, -180.328, 25.778, 195.459, -135.504]
  MoveL 1574 to (94.73, -135.81, -42.78) mm, rotated rx -74.73 ry 0 rz 34.59 deg; joints [-1.953, -87.923, 124.92, -180.938, 25.778, 195.959, -134.433]
  Set speed (1000.0 mm/s)
  MoveL 1575 to (92.71, -135.53, -47.8) mm, rotated rx -74.61 ry 0 rz 34.41 deg; joints [-2.235, -87.783, 124.87, -181.574, 25.778, 196.599, -134.343]
  Set speed (5.0 mm/s)
  MoveL 1576 to (81.81, -119.62, -42.49) mm, rotated rx -74.61 ry 0 rz 34.41 deg; joints [-1.964, -86.994, 125.155, -180.955, 25.778, 196.087, -135.411]
  Set speed (16.7 mm/s)
  MoveL 1577 to (77.51, -122.51, -42.31) mm, rotated rx -74.68 ry 0 rz 32.36 deg; joints [-1.939, -87, 125.154, -180.9, 25.778, 195.97, -133.354]
  MoveL 1578 to (76.94, -122.89, -42.25) mm, rotated rx -74.7 ry 0 rz 32.15 deg; joints [-1.932, -86.99, 125.143, -180.883, 25.778, 195.937, -133.146]
  MoveL 1579 to (72.84, -125.43, -42.04) mm, rotated rx -74.78 ry 0 rz 30.19 deg; joints [-1.903, -87.007, 125.15, -180.818, 25.778, 195.799, -131.177]
  MoveL 1580 to (72.06, -125.92, -41.94) mm, rotated rx -74.82 ry 0 rz 29.91 deg; joints [-1.89, -86.995, 125.135, -180.789, 25.778, 195.741, -130.893]
  MoveL 1581 to (66.64, -129.33, -40.5) mm, rotated rx -75.37 ry 0 rz 27.48 deg; joints [-1.699, -87.018, 125.105, -180.362, 25.778, 194.846, -128.413]
  MoveL 1582 to (63.46, -130.9, -40.56) mm, rotated rx -75.37 ry 0 rz 25.86 deg; joints [-1.703, -87.062, 125.145, -180.369, 25.778, 194.853, -126.782]
  MoveL 1583 to (62.54, -131.38, -40.43) mm, rotated rx -75.41 ry 0 rz 25.63 deg; joints [-1.687, -87.031, 125.113, -180.335, 25.778, 194.786, -126.553]
  MoveL 1584 to (62.02, -131.68, -40.24) mm, rotated rx -75.41 ry 0 rz 25.63 deg; joints [-1.678, -86.988, 125.073, -180.314, 25.778, 194.769, -126.556]
  MoveL 1585 to (56.11, -135.18, -37.23) mm, rotated rx -76.59 ry 0 rz 22.95 deg; joints [-1.272, -87.07, 125.042, -179.401, 25.778, 192.849, -123.761]
  MoveL 1586 to (63.69, -153.09, -41.87) mm, rotated rx -76.59 ry 0 rz 22.95 deg; joints [-1.506, -87.876, 124.767, -179.931, 25.778, 193.276, -122.679]
  Set speed (1000.0 mm/s)
  MoveL 1587 to (68.16, -152.61, -36.11) mm, rotated rx -76.99 ry 0 rz 24.24 deg; joints [-1.126, -87.985, 124.774, -179.074, 25.778, 192.179, -123.876]
  Set speed (5.0 mm/s)
  MoveL 1588 to (60.16, -134.85, -31.61) mm, rotated rx -76.99 ry 0 rz 24.24 deg; joints [-0.9, -87.173, 125.045, -178.566, 25.778, 191.777, -124.962]
  Set speed (16.7 mm/s)
  MoveL 1589 to (61.76, -134.22, -31.26) mm, rotated rx -77.13 ry 0 rz 24.91 deg; joints [-0.853, -87.181, 125.04, -178.46, 25.778, 191.555, -125.617]
  MoveL 1590 to (62.6, -133.84, -31.24) mm, rotated rx -77.13 ry 0 rz 24.91 deg; joints [-0.852, -87.251, 125.101, -178.456, 25.778, 191.552, -125.608]
  MoveL 1591 to (63.41, -133.42, -31.39) mm, rotated rx -77.07 ry 0 rz 25.26 deg; joints [-0.872, -87.247, 125.103, -178.501, 25.778, 191.645, -125.967]
  MoveL 1592 to (70.32, -129.46, -33.2) mm, rotated rx -76.39 ry 0 rz 28.77 deg; joints [-1.11, -87.126, 125.052, -179.038, 25.778, 192.758, -129.543]
  MoveL 1593 to (72.05, -128.64, -32.68) mm, rotated rx -76.59 ry 0 rz 29.52 deg; joints [-1.04, -87.139, 125.046, -178.881, 25.778, 192.429, -130.269]
  MoveL 1594 to (72.71, -128.29, -32.59) mm, rotated rx -76.59 ry 0 rz 29.52 deg; joints [-1.035, -87.196, 125.095, -178.87, 25.778, 192.42, -130.26]
  MoveL 1595 to (73.24, -127.99, -32.6) mm, rotated rx -76.58 ry 0 rz 29.75 deg; joints [-1.038, -87.195, 125.095, -178.875, 25.778, 192.431, -130.497]
  MoveL 1596 to (78.41, -124.63, -33.57) mm, rotated rx -76.22 ry 0 rz 32.02 deg; joints [-1.165, -87.198, 125.128, -179.161, 25.778, 193.026, -132.792]
  MoveL 1597 to (88.71, -141.1, -38.33) mm, rotated rx -76.22 ry 0 rz 32.02 deg; joints [-1.406, -88.004, 124.855, -179.704, 25.778, 193.462, -131.711]
  Set speed (1000.0 mm/s)
  MoveL 1598 to (102.21, -137.05, -2.99) mm, rotated rx -89.52 ry 0 rz 36.06 deg; joints [3.318, -88.221, 124.325, -168.976, 25.778, 171.363, -135.38]
  Set speed (5.0 mm/s)
  MoveL 1599 to (90.44, -120.88, -2.82) mm, rotated rx -89.52 ry 0 rz 36.06 deg; joints [3.304, -87.392, 124.605, -169.048, 25.778, 171.516, -136.481]
  Set speed (16.7 mm/s)
  MoveL 1600 to (88.38, -122.31, -6) mm, rotated rx -88.31 ry 0 rz 35.11 deg; joints [2.877, -87.404, 124.605, -169.971, 25.629, 173.463, -135.607]
  MoveL 1601 to (87.92, -122.62, -6.51) mm, rotated rx -88.31 ry 0 rz 35.11 deg; joints [2.849, -87.366, 124.574, -170.035, 25.629, 173.516, -135.61]
  MoveL 1602 to (87.39, -122.97, -6.95) mm, rotated rx -88.15 ry 0 rz 34.86 deg; joints [2.79, -87.367, 124.574, -170.163, 25.608, 173.784, -135.377]
  MoveL 1603 to (86.92, -123.29, -7.24) mm, rotated rx -88.15 ry 0 rz 34.86 deg; joints [2.773, -87.326, 124.54, -170.202, 25.608, 173.817, -135.381]
  MoveL 1604 to (84.87, -124.65, -8.12) mm, rotated rx -87.81 ry 0 rz 33.93 deg; joints [2.655, -87.327, 124.54, -170.46, 25.569, 174.358, -134.473]
  MoveL 1605 to (83.39, -125.52, -9.9) mm, rotated rx -86.9 ry 0 rz 32.92 deg; joints [2.364, -87.363, 124.54, -171.062, 25.36, 175.751, -133.595]
  MoveL 1606 to (82.93, -125.79, -10.4) mm, rotated rx -86.82 ry 0 rz 32.83 deg; joints [2.319, -87.343, 124.527, -171.165, 25.36, 175.92, -133.513]
  MoveL 1607 to (80.75, -127.03, -12.24) mm, rotated rx -86.11 ry 0 rz 31.88 deg; joints [2.071, -87.343, 124.539, -171.72, 25.305, 177.072, -132.598]
  MoveL 1608 to (80.17, -127.36, -12.59) mm, rotated rx -86.11 ry 0 rz 31.88 deg; joints [2.051, -87.294, 124.498, -171.767, 25.305, 177.11, -132.604]
  MoveL 1609 to (79.49, -127.77, -12.82) mm, rotated rx -86.07 ry 0 rz 31.75 deg; joints [2.028, -87.261, 124.472, -171.819, 25.305, 177.197, -132.478]
  MoveL 1610 to (77.53, -128.92, -13.15) mm, rotated rx -85.95 ry 0 rz 30.88 deg; joints [1.984, -87.261, 124.476, -171.919, 25.299, 177.404, -131.618]
  MoveL 1611 to (77.4, -129, -13.17) mm, rotated rx -85.63 ry 0 rz 30.26 deg; joints [1.915, -87.319, 124.476, -172.024, 25.097, 177.797, -131.127]
  MoveL 1612 to (75.72, -129.77, -15.23) mm, rotated rx -84.84 ry 0 rz 29.55 deg; joints [1.638, -87.319, 124.5, -172.655, 25.061, 179.096, -130.455]
  MoveL 1613 to (74.7, -130.28, -15.95) mm, rotated rx -84.84 ry 0 rz 29.55 deg; joints [1.599, -87.235, 124.432, -172.748, 25.061, 179.172, -130.466]
  MoveL 1614 to (74.3, -130.49, -16.09) mm, rotated rx -84.79 ry 0 rz 29.38 deg; joints [1.58, -87.235, 124.434, -172.791, 25.06, 179.26, -130.294]
  MoveL 1615 to (73.34, -131.02, -16.17) mm, rotated rx -84.79 ry 0 rz 29.38 deg; joints [1.573, -87.153, 124.363, -172.808, 25.06, 179.275, -130.304]
  MoveL 1616 to (72.39, -131.56, -16.01) mm, rotated rx -84.85 ry 0 rz 28.96 deg; joints [1.594, -87.153, 124.361, -172.759, 25.062, 179.173, -129.885]
  MoveL 1617 to (72.28, -131.59, -16.02) mm, rotated rx -84.17 ry 0 rz 27.86 deg; joints [1.447, -87.253, 124.361, -173.008, 24.687, 180.041, -129.05]
  MoveL 1618 to (71.42, -131.71, -18.79) mm, rotated rx -83.11 ry 0 rz 27.55 deg; joints [1.076, -87.253, 124.415, -173.881, 24.685, 181.815, -128.761]
  MoveL 1619 to (71.39, -131.76, -18.67) mm, rotated rx -82.23 ry 0 rz 27.77 deg; joints [0.888, -87.203, 124.4, -174.323, 24.685, 183.061, -128.997]
  MoveL 1620 to (72.97, -130.61, -20.61) mm, rotated rx -81.49 ry 0 rz 28.51 deg; joints [0.628, -87.195, 124.436, -174.931, 24.685, 184.3, -129.761]
  MoveL 1621 to (73.3, -130.32, -21.19) mm, rotated rx -81.49 ry 0 rz 28.51 deg; joints [0.599, -87.209, 124.436, -174.99, 24.626, 184.346, -129.805]
  MoveL 1622 to (73.51, -130.11, -21.78) mm, rotated rx -81.38 ry 0 rz 28.57 deg; joints [0.546, -87.209, 124.437, -175.109, 24.6, 184.548, -129.885]
  MoveL 1623 to (73.91, -129.59, -23.41) mm, rotated rx -80.76 ry 0 rz 28.79 deg; joints [0.328, -87.196, 124.465, -175.622, 24.6, 185.592, -130.142]
  MoveL 1624 to (73.94, -129.56, -23.52) mm, rotated rx -80.1 ry 0 rz 29.59 deg; joints [0.176, -87.032, 124.35, -175.979, 24.6, 186.544, -130.98]
  MoveL 1625 to (75.23, -128.78, -23.7) mm, rotated rx -80.03 ry 0 rz 30.17 deg; joints [0.151, -87.03, 124.353, -176.038, 24.6, 186.664, -131.562]
  MoveL 1626 to (75.71, -128.49, -23.8) mm, rotated rx -80 ry 0 rz 30.32 deg; joints [0.14, -87.041, 124.364, -176.064, 24.598, 186.714, -131.716]
  MoveL 1627 to (77.54, -127.24, -24.56) mm, rotated rx -79.75 ry 0 rz 31.03 deg; joints [0.047, -87.061, 124.4, -176.281, 24.597, 187.144, -132.433]
  MoveL 1628 to (79.37, -126.18, -24.21) mm, rotated rx -79.84 ry 0 rz 32.32 deg; joints [0.084, -87.017, 124.399, -176.216, 24.754, 187.005, -133.606]
  MoveL 1629 to (79.85, -125.89, -24.17) mm, rotated rx -79.84 ry 0 rz 32.42 deg; joints [0.087, -87.038, 124.417, -176.208, 24.754, 186.994, -133.712]
  MoveL 1630 to (80.62, -125.37, -24.31) mm, rotated rx -79.84 ry 0 rz 32.42 deg; joints [0.082, -87.104, 124.473, -176.22, 24.744, 187.003, -133.712]
  MoveL 1631 to (84.37, -122.54, -25.92) mm, rotated rx -79.22 ry 0 rz 34.23 deg; joints [-0.135, -87.084, 124.498, -176.726, 24.744, 188.039, -135.552]
  MoveL 1632 to (85.93, -121.52, -25.55) mm, rotated rx -79.33 ry 0 rz 35.45 deg; joints [-0.094, -87.038, 124.498, -176.65, 24.911, 187.873, -136.651]
  MoveL 1633 to (85.95, -121.5, -25.53) mm, rotated rx -79.99 ry 0 rz 36.19 deg; joints [0.051, -86.982, 124.498, -176.349, 25.174, 186.971, -137.197]
  MoveL 1634 to (87.01, -121.36, -22.54) mm, rotated rx -81.14 ry 0 rz 36.55 deg; joints [0.451, -87.012, 124.449, -175.427, 25.173, 185.072, -137.501]
  MoveL 1635 to (87.23, -121.31, -21.95) mm, rotated rx -81.33 ry 0 rz 36.62 deg; joints [0.523, -87.019, 124.442, -175.261, 25.173, 184.742, -137.561]
  MoveL 1636 to (87.97, -120.98, -20.84) mm, rotated rx -81.33 ry 0 rz 36.62 deg; joints [0.581, -87.081, 124.487, -175.128, 25.173, 184.633, -137.547]
  MoveL 1637 to (90.1, -119.71, -18.88) mm, rotated rx -82.08 ry 0 rz 37.56 deg; joints [0.843, -87.092, 124.452, -174.524, 25.173, 183.392, -138.462]
  MoveL 1638 to (90.09, -119.72, -18.86) mm, rotated rx -82.81 ry 0 rz 37.92 deg; joints [1.002, -87.07, 124.452, -174.186, 25.327, 182.393, -138.696]
  MoveL 1639 to (90.21, -119.83, -17.57) mm, rotated rx -83.3 ry 0 rz 37.93 deg; joints [1.175, -87.073, 124.428, -173.789, 25.327, 181.576, -138.693]
  MoveL 1640 to (90.47, -119.79, -16.57) mm, rotated rx -83.3 ry 0 rz 37.93 deg; joints [1.226, -87.09, 124.436, -173.672, 25.327, 181.48, -138.688]
  MoveL 1641 to (91.5, -119.19, -15.17) mm, rotated rx -83.41 ry 0 rz 37.98 deg; joints [1.323, -87.169, 124.491, -173.449, 25.327, 181.192, -138.722]
  MoveL 1642 to (92.23, -118.67, -14.67) mm, rotated rx -83.6 ry 0 rz 38.32 deg; joints [1.389, -87.169, 124.482, -173.298, 25.329, 180.88, -139.057]
  MoveL 1643 to (92.16, -118.73, -14.72) mm, rotated rx -84.96 ry 0 rz 38.59 deg; joints [1.687, -87.156, 124.482, -172.66, 25.51, 178.997, -139.189]
  MoveL 1644 to (91.86, -119.04, -14.06) mm, rotated rx -85.06 ry 0 rz 38.52 deg; joints [1.74, -87.149, 124.482, -172.548, 25.555, 178.814, -139.089]
  MoveL 1645 to (91.17, -119.81, -11.87) mm, rotated rx -85.89 ry 0 rz 38.13 deg; joints [2.035, -87.149, 124.458, -171.887, 25.598, 177.442, -138.663]
  MoveL 1646 to (91.03, -119.98, -11.18) mm, rotated rx -85.96 ry 0 rz 38.11 deg; joints [2.085, -87.143, 124.458, -171.783, 25.634, 177.289, -138.622]
  MoveL 1647 to (91.3, -119.93, -9.43) mm, rotated rx -85.96 ry 0 rz 38.11 deg; joints [2.174, -87.157, 124.459, -171.58, 25.634, 177.123, -138.62]
  MoveL 1648 to (93.2, -118.68, -5.31) mm, rotated rx -87.53 ry 0 rz 38.97 deg; joints [2.727, -87.157, 124.452, -170.371, 25.797, 174.584, -139.377]
  MoveL 1649 to (93.25, -118.66, -5.43) mm, rotated rx -88.75 ry 0 rz 38.65 deg; joints [2.993, -87.196, 124.461, -169.765, 25.797, 172.864, -139.062]
  MoveL 1650 to (92.38, -119.37, -4.75) mm, rotated rx -89.01 ry 0 rz 38.22 deg; joints [3.084, -87.194, 124.461, -169.57, 25.829, 172.451, -138.618]
  MoveL 1651 to (91.89, -119.77, -4.25) mm, rotated rx -89.1 ry 0 rz 38.11 deg; joints [3.129, -87.179, 124.461, -169.487, 25.886, 172.292, -138.471]
  MoveL 1652 to (90.37, -120.94, -2.83) mm, rotated rx -89.69 ry 0 rz 37.34 deg; joints [3.33, -87.176, 124.461, -169.05, 25.942, 171.359, -137.67]
  MoveL 1653 to (102.5, -136.84, -2.93) mm, rotated rx -89.69 ry 0 rz 37.34 deg; joints [3.348, -88.008, 124.183, -168.972, 25.942, 171.199, -136.569]
  Set speed (1000.0 mm/s)
  MoveL 1654 to (69.67, -151.25, 38.86) mm, rotated rx -103.85 ry 0 rz 25.19 deg; joints [8.547, -87.038, 124.183, -158.766, 28.404, 149.017, -124.044]
  Set speed (5.0 mm/s)
  MoveL 1655 to (61.4, -133.67, 34.08) mm, rotated rx -103.85 ry 0 rz 25.19 deg; joints [8.237, -86.129, 124.183, -159.06, 27.716, 149.371, -125.558]
  Set speed (16.7 mm/s)
  MoveL 1656 to (60.3, -134, 34.77) mm, rotated rx -104.12 ry 0 rz 24.74 deg; joints [8.328, -86.098, 124.183, -158.897, 27.768, 148.981, -125.117]
  MoveL 1657 to (60.33, -134.01, 34.7) mm, rotated rx -104.01 ry 0 rz 23.61 deg; joints [8.329, -86.322, 124.377, -158.891, 27.768, 149.076, -123.956]
  MoveL 1658 to (56.93, -136.29, 31.42) mm, rotated rx -102.74 ry 0 rz 22.05 deg; joints [7.897, -86.462, 124.377, -159.677, 27.526, 150.933, -122.381]
  MoveL 1659 to (56.94, -136.29, 31.37) mm, rotated rx -101.33 ry 0 rz 21.98 deg; joints [7.595, -86.56, 124.374, -160.218, 27.333, 152.747, -122.332]
  MoveL 1660 to (60.3, -135.6, 27.99) mm, rotated rx -100.02 ry 0 rz 23.29 deg; joints [7.145, -86.686, 124.373, -161.063, 27.094, 154.698, -123.639]
  MoveL 1661 to (61.36, -135.26, 27.32) mm, rotated rx -99.64 ry 0 rz 23.86 deg; joints [7.028, -86.701, 124.373, -161.313, 27.078, 155.277, -124.182]
  MoveL 1662 to (62.08, -135.09, 26.55) mm, rotated rx -99.64 ry 0 rz 23.86 deg; joints [6.991, -86.74, 124.373, -161.329, 26.971, 155.279, -124.243]
  MoveL 1663 to (69.88, -133.18, 13.65) mm, rotated rx -94.69 ry 0 rz 26.87 deg; joints [5.268, -87.091, 124.374, -164.737, 26.137, 162.87, -127.361]
  MoveL 1664 to (70.2, -133.1, 12.83) mm, rotated rx -94.69 ry 0 rz 26.87 deg; joints [5.227, -87.11, 124.374, -164.801, 26.081, 162.918, -127.391]
  MoveL 1665 to (69.89, -133.43, 10.9) mm, rotated rx -94.69 ry 0 rz 26.87 deg; joints [5.128, -87.105, 124.37, -165.026, 26.081, 163.099, -127.371]
  MoveL 1666 to (69.52, -133.67, 10.31) mm, rotated rx -94.47 ry 0 rz 26.71 deg; joints [5.049, -87.116, 124.37, -165.189, 26.046, 163.454, -127.216]
  MoveL 1667 to (68.72, -134.14, 9.53) mm, rotated rx -94.47 ry 0 rz 26.71 deg; joints [5.004, -87.059, 124.319, -165.29, 26.046, 163.537, -127.214]
  MoveL 1668 to (62.93, -137.14, 6.34) mm, rotated rx -93.26 ry 0 rz 24.23 deg; joints [4.578, -87.112, 124.319, -166.176, 25.863, 165.45, -124.785]
  MoveL 1669 to (62.6, -137.3, 6.11) mm, rotated rx -93.14 ry 0 rz 24.03 deg; joints [4.54, -87.123, 124.319, -166.246, 25.827, 165.626, -124.597]
  MoveL 1670 to (57.66, -139.56, 2.56) mm, rotated rx -91.77 ry 0 rz 21.93 deg; joints [4.059, -87.173, 124.319, -167.254, 25.62, 167.798, -122.573]
  MoveL 1671 to (65.13, -158.1, 3.18) mm, rotated rx -91.77 ry 0 rz 21.93 deg; joints [4.116, -87.987, 124.023, -167.077, 25.621, 167.543, -121.482]
  Set speed (1000.0 mm/s)
  MoveL 1672 to (61.23, -159.61, 4.89) mm, rotated rx -91.82 ry 0 rz 21.81 deg; joints [4.208, -87.829, 124.02, -167.077, 26.093, 167.522, -121.047]
  Set speed (5.0 mm/s)
  MoveL 1673 to (53.8, -141.05, 4.25) mm, rotated rx -91.82 ry 0 rz 21.81 deg; joints [4.15, -87.007, 124.31, -167.255, 26.093, 167.779, -122.139]
  Set speed (16.7 mm/s)
  MoveL 1674 to (53.45, -141.12, 5.86) mm, rotated rx -92.43 ry 0 rz 21.67 deg; joints [4.365, -86.986, 124.309, -166.806, 26.179, 166.812, -121.975]
  MoveL 1675 to (53.42, -141.12, 5.84) mm, rotated rx -93.06 ry 0 rz 21.16 deg; joints [4.509, -87.052, 124.363, -166.48, 26.179, 165.913, -121.484]
  MoveL 1676 to (50.11, -142.26, 7.61) mm, rotated rx -93.74 ry 0 rz 19.83 deg; joints [4.746, -87.026, 124.363, -165.99, 26.279, 164.853, -120.122]
  MoveL 1677 to (49.43, -142.47, 8.08) mm, rotated rx -93.84 ry 0 rz 19.69 deg; joints [4.791, -87.007, 124.364, -165.916, 26.338, 164.696, -119.949]
  MoveL 1678 to (46.88, -143.14, 10.85) mm, rotated rx -94.76 ry 0 rz 18.83 deg; joints [5.132, -86.945, 124.364, -165.242, 26.531, 163.243, -119.024]
  MoveL 1679 to (43.15, -144.21, 12.26) mm, rotated rx -95.55 ry 0 rz 16.99 deg; joints [5.378, -86.949, 124.367, -164.691, 26.531, 162.013, -117.229]
  MoveL 1680 to (42.56, -144.35, 12.56) mm, rotated rx -95.61 ry 0 rz 16.88 deg; joints [5.405, -86.932, 124.367, -164.657, 26.582, 161.933, -117.093]
  MoveL 1681 to (42.42, -144.38, 12.73) mm, rotated rx -95.12 ry 0 rz 15.47 deg; joints [5.319, -87.115, 124.416, -164.657, 26.207, 162.38, -115.912]
  MoveL 1682 to (42.22, -144.5, 11.97) mm, rotated rx -94.8 ry 0 rz 15.37 deg; joints [5.209, -87.133, 124.416, -164.88, 26.154, 162.884, -115.83]
  MoveL 1683 to (41.24, -145.04, 8.08) mm, rotated rx -93.32 ry 0 rz 14.96 deg; joints [4.688, -87.202, 124.416, -165.953, 25.927, 165.208, -115.473]
  MoveL 1684 to (41.22, -145.05, 8.08) mm, rotated rx -92.4 ry 0 rz 15.19 deg; joints [4.484, -87.202, 124.42, -166.42, 25.926, 166.511, -115.674]
  MoveL 1685 to (42.7, -144.71, 6.56) mm, rotated rx -91.82 ry 0 rz 15.77 deg; joints [4.28, -87.223, 124.42, -166.847, 25.843, 167.428, -116.275]
  MoveL 1686 to (43.29, -144.57, 5.76) mm, rotated rx -91.64 ry 0 rz 15.9 deg; joints [4.199, -87.241, 124.42, -167.002, 25.777, 167.733, -116.438]
  MoveL 1687 to (45.2, -144.07, 2.42) mm, rotated rx -90.03 ry 0 rz 17.09 deg; joints [3.675, -87.241, 124.435, -168.186, 25.738, 170.298, -117.592]
  MoveL 1688 to (47.5, -143.35, 1.53) mm, rotated rx -89.69 ry 0 rz 18 deg; joints [3.554, -87.248, 124.435, -168.444, 25.693, 170.847, -118.525]
  MoveL 1689 to (48.44, -143.04, 0.99) mm, rotated rx -89.56 ry 0 rz 18.23 deg; joints [3.498, -87.267, 124.435, -168.546, 25.626, 171.06, -118.796]
  MoveL 1690 to (53.7, -141.11, -3.5) mm, rotated rx -87.93 ry 0 rz 20.24 deg; joints [2.912, -87.298, 124.435, -169.803, 25.379, 173.692, -120.932]
  MoveL 1691 to (54.37, -140.82, -4.48) mm, rotated rx -87.93 ry 0 rz 20.24 deg; joints [2.864, -87.328, 124.435, -169.878, 25.275, 173.747, -121]
  MoveL 1692 to (54.55, -140.74, -4.93) mm, rotated rx -87.76 ry 0 rz 20.31 deg; joints [2.803, -87.329, 124.435, -170.011, 25.254, 174.026, -121.084]
  MoveL 1693 to (54.71, -140.65, -5.7) mm, rotated rx -87.76 ry 0 rz 20.31 deg; joints [2.764, -87.337, 124.435, -170.089, 25.219, 174.087, -121.106]
  MoveL 1694 to (54.93, -140.34, -9.65) mm, rotated rx -86.26 ry 0 rz 20.43 deg; joints [2.232, -87.337, 124.443, -171.274, 25.06, 176.551, -121.325]
  MoveL 1695 to (56.36, -139.38, -14.28) mm, rotated rx -84.26 ry 0 rz 21.12 deg; joints [1.558, -87.337, 124.506, -172.824, 24.989, 179.817, -122.074]
  MoveL 1696 to (63.53, -157.94, -16.28) mm, rotated rx -84.26 ry 0 rz 21.12 deg; joints [1.471, -88.162, 124.23, -173.002, 24.989, 179.903, -120.967]
  Set speed (1000.0 mm/s)
  MoveL 1697 to (46.92, -164.25, -8.17) mm, rotated rx -87.45 ry 0 rz 16.76 deg; joints [2.587, -88.013, 124.23, -170.682, 25.878, 174.833, -115.991]
  Set speed (5.0 mm/s)
  MoveL 1698 to (41.16, -145.12, -7.28) mm, rotated rx -87.45 ry 0 rz 16.76 deg; joints [2.612, -87.174, 124.501, -170.657, 25.878, 174.894, -117.098]
  Set speed (16.7 mm/s)
  MoveL 1699 to (40.47, -145.44, -4.09) mm, rotated rx -88.66 ry 0 rz 16.48 deg; joints [3.041, -87.169, 124.501, -169.735, 26.023, 172.942, -116.73]
  MoveL 1700 to (37.19, -146.37, -0.4) mm, rotated rx -90.49 ry 0 rz 14.95 deg; joints [3.632, -87.169, 124.501, -168.453, 26.165, 170.083, -115.155]
  MoveL 1701 to (37.63, -146.26, -0.79) mm, rotated rx -90.49 ry 0 rz 14.95 deg; joints [3.613, -87.189, 124.501, -168.472, 26.104, 170.095, -115.196]
  MoveL 1702 to (37.24, -146.36, -0.52) mm, rotated rx -90.59 ry 0 rz 14.8 deg; joints [3.649, -87.187, 124.501, -168.396, 26.117, 169.933, -115.037]
  MoveL 1703 to (33.99, -147.13, 2.15) mm, rotated rx -91.55 ry 0 rz 13.6 deg; joints [3.996, -87.156, 124.501, -167.675, 26.271, 168.395, -113.768]
  MoveL 1704 to (33.07, -147.3, 4.06) mm, rotated rx -91.55 ry 0 rz 13.6 deg; joints [4.092, -87.11, 124.501, -167.524, 26.421, 168.282, -113.677]
  MoveL 1705 to (33.05, -147.29, 4.63) mm, rotated rx -91.77 ry 0 rz 13.6 deg; joints [4.169, -87.103, 124.501, -167.364, 26.452, 167.937, -113.663]
  MoveL 1706 to (33.65, -146.86, 10.18) mm, rotated rx -93.75 ry 0 rz 13.85 deg; joints [4.883, -87.025, 124.501, -165.9, 26.745, 164.805, -113.825]
  MoveL 1707 to (33.31, -146.88, 11.08) mm, rotated rx -94.53 ry 0 rz 13.67 deg; joints [5.102, -87.001, 124.501, -165.451, 26.825, 163.661, -113.635]
  MoveL 1708 to (33.12, -146.86, 11.95) mm, rotated rx -94.66 ry 0 rz 13.65 deg; joints [5.173, -86.985, 124.501, -165.316, 26.872, 163.431, -113.601]
  MoveL 1709 to (32.94, -146.65, 14.63) mm, rotated rx -95.61 ry 0 rz 13.61 deg; joints [5.515, -86.931, 124.501, -164.636, 27.028, 161.953, -113.523]
  MoveL 1710 to (31.71, -146.74, 16.44) mm, rotated rx -96.77 ry 0 rz 12.99 deg; joints [5.862, -86.886, 124.501, -163.929, 27.141, 160.23, -112.91]
  MoveL 1711 to (31.44, -146.74, 16.89) mm, rotated rx -96.86 ry 0 rz 12.94 deg; joints [5.905, -86.872, 124.501, -163.854, 27.176, 160.081, -112.842]
  MoveL 1712 to (30.13, -146.72, 19.3) mm, rotated rx -97.78 ry 0 rz 12.45 deg; joints [6.226, -86.808, 124.501, -163.23, 27.331, 158.678, -112.335]
  MoveL 1713 to (29.8, -146.69, 20.02) mm, rotated rx -97.98 ry 0 rz 12.37 deg; joints [6.305, -86.787, 124.501, -163.083, 27.381, 158.366, -112.239]
  MoveL 1714 to (28.15, -146.67, 22.3) mm, rotated rx -99.02 ry 0 rz 11.66 deg; joints [6.645, -86.719, 124.501, -162.417, 27.521, 156.812, -111.534]
  MoveL 1715 to (28.2, -146.65, 22.33) mm, rotated rx -99.35 ry 0 rz 10.46 deg; joints [6.74, -86.924, 124.686, -162.208, 27.521, 156.312, -110.337]
  MoveL 1716 to (24.5, -147.61, 20.46) mm, rotated rx -98.63 ry 0 rz 9 deg; joints [6.49, -86.983, 124.686, -162.684, 27.396, 157.396, -108.887]
  MoveL 1717 to (23.28, -147.84, 20.2) mm, rotated rx -98.63 ry 0 rz 9 deg; joints [6.469, -86.897, 124.609, -162.732, 27.396, 157.436, -108.891]
  MoveL 1718 to (21.71, -148.02, 20.6) mm, rotated rx -98.64 ry 0 rz 8.86 deg; joints [6.483, -86.817, 124.556, -162.732, 27.453, 157.435, -108.723]
  MoveL 1719 to (19.07, -148.15, 22.25) mm, rotated rx -99.27 ry 0 rz 7.85 deg; joints [6.703, -86.765, 124.556, -162.314, 27.564, 156.481, -107.702]
  MoveL 1720 to (17.91, -148.03, 23.97) mm, rotated rx -99.27 ry 0 rz 7.85 deg; joints [6.787, -86.699, 124.556, -162.233, 27.741, 156.435, -107.605]
  MoveL 1721 to (17.88, -147.83, 25.16) mm, rotated rx -99.37 ry 0 rz 7.83 deg; joints [6.868, -86.68, 124.556, -162.078, 27.778, 156.219, -107.591]
  MoveL 1722 to (18.2, -147.52, 26.66) mm, rotated rx -99.95 ry 0 rz 7.97 deg; joints [7.069, -86.629, 124.556, -161.703, 27.882, 155.352, -107.724]
  MoveL 1723 to (18.27, -147.53, 26.58) mm, rotated rx -100.76 ry 0 rz 7.79 deg; joints [7.238, -86.605, 124.556, -161.351, 27.907, 154.273, -107.584]
  MoveL 1724 to (15.91, -147.31, 29.23) mm, rotated rx -101.78 ry 0 rz 6.9 deg; joints [7.589, -86.506, 124.556, -160.706, 28.095, 152.766, -106.687]
  MoveL 1725 to (15.51, -147.25, 29.72) mm, rotated rx -101.84 ry 0 rz 6.84 deg; joints [7.627, -86.485, 124.556, -160.655, 28.144, 152.669, -106.612]
  MoveL 1726 to (14.83, -147.1, 30.8) mm, rotated rx -102.26 ry 0 rz 6.59 deg; joints [7.77, -86.442, 124.556, -160.396, 28.223, 152.057, -106.355]
  MoveL 1727 to (12.15, -147.03, 32.27) mm, rotated rx -103.16 ry 0 rz 5.2 deg; joints [8.037, -86.395, 124.556, -159.848, 28.263, 150.732, -105.051]
  MoveL 1728 to (11.52, -146.98, 32.71) mm, rotated rx -103.25 ry 0 rz 5.09 deg; joints [8.077, -86.369, 124.556, -159.801, 28.325, 150.615, -104.912]
  MoveL 1729 to (9.08, -146.59, 35.18) mm, rotated rx -104.12 ry 0 rz 4.26 deg; joints [8.383, -86.255, 124.556, -159.278, 28.529, 149.362, -104.062]
  MoveL 1730 to (8.71, -146.49, 35.65) mm, rotated rx -104.12 ry 0 rz 4.26 deg; joints [8.405, -86.233, 124.556, -159.265, 28.584, 149.359, -104.033]
  MoveL 1731 to (8.05, -146.3, 36.55) mm, rotated rx -104.57 ry 0 rz 3.94 deg; joints [8.545, -86.19, 124.556, -159.007, 28.644, 148.718, -103.735]
  MoveL 1732 to (8.17, -146.3, 36.55) mm, rotated rx -104.87 ry 0 rz 2.79 deg; joints [8.633, -86.376, 124.73, -158.817, 28.644, 148.264, -102.604]
  MoveL 1733 to (6.9, -146.51, 35.99) mm, rotated rx -104.65 ry 0 rz 2.29 deg; joints [8.56, -86.403, 124.73, -158.946, 28.601, 148.577, -102.099]
  MoveL 1734 to (6.1, -146.6, 35.76) mm, rotated rx -104.62 ry 0 rz 2.15 deg; joints [8.538, -86.381, 124.708, -158.993, 28.601, 148.647, -101.952]
  MoveL 1735 to (1.55, -146.87, 35.12) mm, rotated rx -104.39 ry 0 rz 0.47 deg; joints [8.456, -86.399, 124.707, -159.153, 28.58, 149.002, -100.244]
  MoveL 1736 to (0.94, -146.87, 35.12) mm, rotated rx -104.27 ry 0 rz -0.11 deg; joints [8.438, -86.459, 124.738, -159.153, 28.521, 149.107, -99.694]
  MoveL 1737 to (-2.9, -147.33, 33) mm, rotated rx -103.45 ry 0 rz -1.61 deg; joints [8.158, -86.553, 124.738, -159.65, 28.362, 150.298, -98.195]
  MoveL 1738 to (-3.8, -147.5, 32.22) mm, rotated rx -103.16 ry 0 rz -1.92 deg; joints [8.058, -86.582, 124.738, -159.835, 28.319, 150.72, -97.874]
  MoveL 1739 to (-7.46, -147.74, 30.42) mm, rotated rx -102.47 ry 0 rz -3.33 deg; joints [7.821, -86.657, 124.738, -160.263, 28.187, 151.734, -96.46]
  MoveL 1740 to (-11.67, -148.19, 26.67) mm, rotated rx -100.87 ry 0 rz -5.15 deg; joints [7.292, -86.834, 124.738, -161.189, 27.834, 154.018, -94.684]
  MoveL 1741 to (-12.15, -148.21, 26.31) mm, rotated rx -100.79 ry 0 rz -5.26 deg; joints [7.256, -86.834, 124.736, -161.267, 27.834, 154.158, -94.564]
  MoveL 1742 to (-14.84, -148.24, 24.72) mm, rotated rx -100.23 ry 0 rz -6.21 deg; joints [7.055, -86.878, 124.736, -161.655, 27.754, 155.016, -93.602]
  MoveL 1743 to (-16.01, -148.36, 23.23) mm, rotated rx -99.43 ry 0 rz -6.92 deg; joints [6.809, -86.969, 124.736, -162.071, 27.545, 156.124, -92.961]
  MoveL 1744 to (-16.61, -148.38, 22.69) mm, rotated rx -99.43 ry 0 rz -6.92 deg; joints [6.778, -86.936, 124.705, -162.139, 27.545, 156.179, -92.955]
  MoveL 1745 to (-17.21, -148.37, 22.31) mm, rotated rx -99.29 ry 0 rz -7.14 deg; joints [6.727, -86.949, 124.705, -162.236, 27.518, 156.4, -92.731]
  MoveL 1746 to (-21.4, -148.14, 19.91) mm, rotated rx -98.4 ry 0 rz -8.7 deg; joints [6.413, -87.015, 124.705, -162.842, 27.376, 157.756, -91.182]
  MoveL 1747 to (-21.33, -148.15, 20.01) mm, rotated rx -97.44 ry 0 rz -9.13 deg; joints [6.213, -87.107, 124.705, -163.149, 27.134, 158.932, -90.856]
  MoveL 1748 to (-20.58, -148.81, 15.47) mm, rotated rx -95.71 ry 0 rz -8.81 deg; joints [5.605, -87.223, 124.705, -164.344, 26.846, 161.596, -91.221]
  MoveL 1749 to (-20.61, -148.91, 14.47) mm, rotated rx -95.71 ry 0 rz -8.81 deg; joints [5.554, -87.232, 124.707, -164.447, 26.828, 161.677, -91.221]
  MoveL 1750 to (-20.84, -148.95, 13.71) mm, rotated rx -95.59 ry 0 rz -8.84 deg; joints [5.49, -87.237, 124.707, -164.583, 26.817, 161.9, -91.188]
  MoveL 1751 to (-21.83, -148.98, 11.55) mm, rotated rx -94.77 ry 0 rz -9.2 deg; joints [5.2, -87.282, 124.707, -165.165, 26.687, 163.18, -90.849]
  MoveL 1752 to (-21.68, -149.16, 9.48) mm, rotated rx -93.52 ry 0 rz -9.22 deg; joints [4.821, -87.343, 124.707, -165.922, 26.497, 165.021, -90.894]
  MoveL 1753 to (-21.88, -149.2, 8.29) mm, rotated rx -93.52 ry 0 rz -9.22 deg; joints [4.76, -87.342, 124.707, -166.057, 26.495, 165.131, -90.885]
  MoveL 1754 to (-22.55, -149.15, 7.3) mm, rotated rx -93.47 ry 0 rz -9.24 deg; joints [4.695, -87.313, 124.683, -166.203, 26.495, 165.304, -90.853]
  MoveL 1755 to (-23.91, -148.99, 6.04) mm, rotated rx -92.99 ry 0 rz -9.76 deg; joints [4.526, -87.332, 124.683, -166.549, 26.424, 166.055, -90.354]
  MoveL 1756 to (-24.53, -148.93, 4.9) mm, rotated rx -92.35 ry 0 rz -10.16 deg; joints [4.328, -87.371, 124.683, -166.935, 26.29, 166.996, -90.01]
  MoveL 1757 to (-24.97, -148.88, 4.36) mm, rotated rx -92.35 ry 0 rz -10.16 deg; joints [4.299, -87.344, 124.66, -167.001, 26.29, 167.049, -90.009]
  MoveL 1758 to (-25.42, -148.81, 3.98) mm, rotated rx -92.29 ry 0 rz -10.24 deg; joints [4.264, -87.332, 124.651, -167.081, 26.29, 167.181, -89.933]
  MoveL 1759 to (-27.35, -148.5, 2.61) mm, rotated rx -91.77 ry 0 rz -10.98 deg; joints [4.08, -87.348, 124.651, -167.464, 26.217, 168.006, -89.215]
  MoveL 1760 to (-29.2, -148.17, 1.12) mm, rotated rx -91.18 ry 0 rz -11.72 deg; joints [3.875, -87.367, 124.651, -167.889, 26.127, 168.93, -88.509]
  MoveL 1761 to (-30.79, -147.85, 0.61) mm, rotated rx -91.18 ry 0 rz -11.72 deg; joints [3.841, -87.252, 124.551, -167.965, 26.127, 168.993, -88.518]
  MoveL 1762 to (-31.85, -147.62, 0.66) mm, rotated rx -91.2 ry 0 rz -12.14 deg; joints [3.848, -87.252, 124.55, -167.952, 26.13, 168.965, -88.104]
  MoveL 1763 to (-33.74, -147.19, 1.72) mm, rotated rx -91.2 ry 0 rz -12.14 deg; joints [3.897, -87.164, 124.539, -167.933, 26.359, 168.965, -87.955]
  MoveL 1764 to (-39.02, -145.58, 9.53) mm, rotated rx -94.16 ry 0 rz -14.23 deg; joints [4.945, -87.055, 124.539, -165.783, 26.789, 164.297, -85.727]
  MoveL 1765 to (-41.85, -144.54, 12.77) mm, rotated rx -95.49 ry 0 rz -15.45 deg; joints [5.401, -86.996, 124.539, -164.857, 26.965, 162.235, -84.478]
  MoveL 1766 to (-42.19, -144.4, 13.29) mm, rotated rx -95.49 ry 0 rz -15.45 deg; joints [5.427, -86.977, 124.539, -164.828, 27.022, 162.216, -84.445]
  MoveL 1767 to (-42.43, -144.28, 13.77) mm, rotated rx -95.68 ry 0 rz -15.55 deg; joints [5.491, -86.966, 124.539, -164.701, 27.051, 161.933, -84.341]
  MoveL 1768 to (-44.48, -143.1, 18.72) mm, rotated rx -97.52 ry 0 rz -16.4 deg; joints [6.142, -86.843, 124.539, -163.433, 27.365, 159.109, -83.435]
  MoveL 1769 to (-47.27, -141.59, 22.89) mm, rotated rx -99.27 ry 0 rz -17.68 deg; joints [6.733, -86.721, 124.539, -162.287, 27.629, 156.467, -82.14]
  MoveL 1770 to (-47.64, -141.33, 23.72) mm, rotated rx -99.43 ry 0 rz -17.75 deg; joints [6.807, -86.693, 124.54, -162.165, 27.699, 156.222, -82.043]
  MoveL 1771 to (-48.96, -140.12, 27.88) mm, rotated rx -100.98 ry 0 rz -18.36 deg; joints [7.348, -86.549, 124.54, -161.161, 27.987, 153.911, -81.419]
  MoveL 1772 to (-49.1, -139.98, 28.33) mm, rotated rx -101.16 ry 0 rz -18.43 deg; joints [7.41, -86.531, 124.539, -161.046, 28.02, 153.642, -81.346]
  MoveL 1773 to (-50.03, -138.68, 32.76) mm, rotated rx -102.79 ry 0 rz -18.9 deg; joints [7.978, -86.358, 124.542, -160.025, 28.344, 151.253, -80.867]
  MoveL 1774 to (-50.07, -138.48, 33.54) mm, rotated rx -102.88 ry 0 rz -18.91 deg; joints [8.036, -86.336, 124.542, -159.929, 28.387, 151.092, -80.856]
  MoveL 1775 to (-50.26, -138.3, 33.93) mm, rotated rx -103.36 ry 0 rz -19.08 deg; joints [8.158, -86.304, 124.542, -159.694, 28.431, 150.429, -80.701]
  MoveL 1776 to (-50.22, -138.32, 33.9) mm, rotated rx -103.85 ry 0 rz -20.32 deg; joints [8.286, -86.486, 124.717, -159.42, 28.431, 149.721, -79.49]
  MoveL 1777 to (-52.26, -137.77, 33.08) mm, rotated rx -103.53 ry 0 rz -21.14 deg; joints [8.177, -86.523, 124.717, -159.613, 28.37, 150.184, -78.671]
  MoveL 1778 to (-53.42, -137.37, 32.92) mm, rotated rx -103.53 ry 0 rz -21.14 deg; joints [8.159, -86.439, 124.641, -159.653, 28.37, 150.218, -78.674]
  MoveL 1779 to (-54.01, -137.12, 33) mm, rotated rx -103.56 ry 0 rz -21.38 deg; joints [8.169, -86.436, 124.641, -159.636, 28.376, 150.176, -78.425]
  MoveL 1780 to (-55.34, -136.41, 33.71) mm, rotated rx -103.56 ry 0 rz -21.38 deg; joints [8.193, -86.328, 124.569, -159.624, 28.438, 150.176, -78.401]
  MoveL 1781 to (-59.26, -133.49, 38.41) mm, rotated rx -105.4 ry 0 rz -23.23 deg; joints [8.813, -86.109, 124.569, -158.538, 28.796, 147.546, -76.575]
  MoveL 1782 to (-59.52, -133.29, 38.71) mm, rotated rx -105.54 ry 0 rz -23.38 deg; joints [8.856, -86.095, 124.569, -158.458, 28.815, 147.348, -76.434]
  MoveL 1783 to (-64.29, -130.15, 41.64) mm, rotated rx -106.83 ry 0 rz -25.81 deg; joints [9.273, -85.954, 124.569, -157.704, 29, 145.495, -74.078]
  MoveL 1784 to (-64.9, -129.68, 42.18) mm, rotated rx -106.96 ry 0 rz -25.96 deg; joints [9.323, -85.918, 124.569, -157.648, 29.074, 145.342, -73.896]
  MoveL 1785 to (-67.67, -127.47, 44.47) mm, rotated rx -108.06 ry 0 rz -28.11 deg; joints [9.672, -85.861, 124.581, -156.913, 29.074, 143.672, -71.921]
  MoveL 1786 to (-68.58, -127.04, 44.33) mm, rotated rx -108.01 ry 0 rz -28.52 deg; joints [9.653, -85.87, 124.581, -156.945, 29.062, 143.754, -71.518]
  MoveL 1787 to (-69.23, -126.7, 44.28) mm, rotated rx -108 ry 0 rz -28.7 deg; joints [9.646, -85.854, 124.566, -156.959, 29.062, 143.773, -71.332]
  MoveL 1788 to (-73.83, -124.07, 44.3) mm, rotated rx -108.01 ry 0 rz -30.75 deg; joints [9.648, -85.844, 124.559, -156.959, 29.066, 143.766, -69.28]
  MoveL 1789 to (-74.21, -123.86, 44.26) mm, rotated rx -107.99 ry 0 rz -31 deg; joints [9.644, -85.858, 124.567, -156.959, 29.054, 143.781, -69.036]
  MoveL 1790 to (-79.86, -120.38, 44.03) mm, rotated rx -107.9 ry 0 rz -33.59 deg; joints [9.614, -85.867, 124.567, -157.017, 29.048, 143.913, -66.431]
  MoveL 1791 to (-80.54, -119.9, 44.09) mm, rotated rx -107.92 ry 0 rz -33.8 deg; joints [9.618, -85.843, 124.55, -157.017, 29.058, 143.896, -66.225]
  MoveL 1792 to (-84.53, -116.94, 44.58) mm, rotated rx -108.11 ry 0 rz -35.76 deg; joints [9.682, -85.814, 124.55, -156.912, 29.1, 143.629, -64.266]
  MoveL 1793 to (-95.84, -132.21, 50.82) mm, rotated rx -108.12 ry 0 rz -35.86 deg; joints [10.075, -86.683, 124.55, -156.536, 29.862, 143.196, -62.652]
  Set speed (1000.0 mm/s)
  MoveL 1794 to (-98.33, -130.06, 51.52) mm, rotated rx -108.35 ry 0 rz -36.87 deg; joints [10.154, -86.629, 124.55, -156.44, 29.96, 142.911, -61.617]
  Set speed (5.0 mm/s)
  MoveL 1795 to (-86.94, -114.87, 45.23) mm, rotated rx -108.35 ry 0 rz -36.87 deg; joints [9.761, -85.762, 124.55, -156.812, 29.193, 143.332, -63.136]
  Set speed (16.7 mm/s)
  MoveL 1796 to (-87.73, -114.16, 45.49) mm, rotated rx -108.45 ry 0 rz -37.29 deg; joints [9.795, -85.747, 124.55, -156.755, 29.215, 143.187, -62.72]
  MoveL 1797 to (-99.22, -129.26, 51.82) mm, rotated rx -108.45 ry 0 rz -37.29 deg; joints [10.191, -86.613, 124.55, -156.382, 29.984, 142.765, -61.201]
  Set speed (1000.0 mm/s)
  MoveL 1798 to (-108.79, -120.03, 54.78) mm, rotated rx -109.49 ry 0 rz -41.96 deg; joints [10.55, -86.448, 124.55, -155.81, 30.221, 141.323, -56.556]
  Set speed (5.0 mm/s)
  MoveL 1799 to (-96.18, -106.01, 48.11) mm, rotated rx -109.49 ry 0 rz -41.96 deg; joints [10.136, -85.594, 124.55, -156.194, 29.428, 141.753, -58.08]
  Set speed (16.7 mm/s)
  MoveL 1800 to (-99.42, -102.43, 49.31) mm, rotated rx -109.98 ry 0 rz -43.89 deg; joints [10.292, -85.521, 124.55, -155.94, 29.528, 141.096, -56.172]
  MoveL 1801 to (-100.01, -101.64, 49.73) mm, rotated rx -110.06 ry 0 rz -44.06 deg; joints [10.329, -85.481, 124.55, -155.927, 29.615, 141.011, -55.954]
  MoveL 1802 to (-101.98, -98.93, 51.18) mm, rotated rx -110.67 ry 0 rz -45.44 deg; joints [10.521, -85.393, 124.55, -155.608, 29.723, 140.186, -54.61]
  MoveL 1803 to (-102.57, -97.95, 51.87) mm, rotated rx -110.86 ry 0 rz -45.73 deg; joints [10.592, -85.34, 124.55, -155.529, 29.818, 139.951, -54.3]
  MoveL 1804 to (-104.87, -93.14, 55.92) mm, rotated rx -112.45 ry 0 rz -47.72 deg; joints [11.105, -85.067, 124.55, -154.736, 30.17, 137.829, -52.372]
  MoveL 1805 to (-104.81, -93.16, 56.04) mm, rotated rx -111.29 ry 0 rz -49.24 deg; joints [10.895, -85.345, 124.558, -154.736, 29.595, 138.897, -51.136]
  MoveL 1806 to (-104.67, -93.92, 55.05) mm, rotated rx -110.88 ry 0 rz -48.97 deg; joints [10.766, -85.412, 124.558, -154.942, 29.513, 139.442, -51.385]
  MoveL 1807 to (-104.54, -94.17, 54.86) mm, rotated rx -110.64 ry 0 rz -48.72 deg; joints [10.708, -85.427, 124.558, -155.064, 29.513, 139.771, -51.595]
  MoveL 1808 to (-102.34, -98.93, 50.44) mm, rotated rx -108.57 ry 0 rz -46.01 deg; joints [10.066, -85.662, 124.557, -156.255, 29.31, 142.709, -54.075]
  MoveL 1809 to (-101.03, -100.32, 50.38) mm, rotated rx -108.54 ry 0 rz -45.24 deg; joints [10.057, -85.666, 124.557, -156.27, 29.305, 142.747, -54.844]
  MoveL 1810 to (-100.46, -100.97, 50.2) mm, rotated rx -108.54 ry 0 rz -45.24 deg; joints [10.057, -85.733, 124.615, -156.268, 29.305, 142.744, -54.835]
  MoveL 1811 to (-99.81, -102.26, 48.86) mm, rotated rx -108.54 ry 0 rz -45.24 deg; joints [10.001, -85.838, 124.656, -156.296, 29.179, 142.744, -54.887]
  MoveL 1812 to (-99.79, -102.49, 48.42) mm, rotated rx -108.38 ry 0 rz -45.18 deg; joints [9.946, -85.864, 124.656, -156.383, 29.142, 142.961, -54.947]
  MoveL 1813 to (-99.7, -103.53, 46.31) mm, rotated rx -107.54 ry 0 rz -44.86 deg; joints [9.67, -85.984, 124.656, -156.843, 28.971, 144.125, -55.237]
  MoveL 1814 to (-99.77, -103.45, 46.33) mm, rotated rx -107 ry 0 rz -43.55 deg; joints [9.531, -85.808, 124.478, -157.14, 28.971, 144.895, -56.497]
  MoveL 1815 to (-96.16, -106, 48.23) mm, rotated rx -107.76 ry 0 rz -41.8 deg; joints [9.78, -85.701, 124.478, -156.723, 29.125, 143.843, -58.272]
  MoveL 1816 to (-108.85, -120.19, 54.33) mm, rotated rx -107.76 ry 0 rz -41.8 deg; joints [10.164, -86.572, 124.478, -156.37, 29.889, 143.436, -56.75]
  Set speed (1000.0 mm/s)
  MoveL 1817 to (-95.78, -132.54, 50.07) mm, rotated rx -106.41 ry 0 rz -36.45 deg; joints [9.682, -86.892, 124.478, -156.934, 29.262, 145.131, -62.294]
  Set speed (5.0 mm/s)
  MoveL 1818 to (-84.39, -117.1, 44.42) mm, rotated rx -106.41 ry 0 rz -36.45 deg; joints [9.323, -86.009, 124.478, -157.264, 28.521, 145.518, -63.814]
  Set speed (16.7 mm/s)
  MoveL 1819 to (-81.74, -120.21, 40.93) mm, rotated rx -105.02 ry 0 rz -34.88 deg; joints [8.861, -86.189, 124.478, -158.064, 28.247, 147.482, -65.352]
  MoveL 1820 to (-81.42, -121.13, 38.81) mm, rotated rx -105.02 ry 0 rz -34.88 deg; joints [8.758, -86.26, 124.478, -158.18, 28.093, 147.551, -65.413]
  MoveL 1821 to (-82.02, -121.15, 37.44) mm, rotated rx -104.91 ry 0 rz -34.9 deg; joints [8.665, -86.276, 124.478, -158.381, 28.092, 147.822, -65.355]
  MoveL 1822 to (-84.98, -120.27, 33.5) mm, rotated rx -103.37 ry 0 rz -36.03 deg; joints [8.146, -86.454, 124.478, -159.31, 27.796, 150.042, -64.199]
  MoveL 1823 to (-85.5, -120.05, 32.94) mm, rotated rx -103.3 ry 0 rz -36.12 deg; joints [8.1, -86.451, 124.47, -159.41, 27.796, 150.196, -64.096]
  MoveL 1824 to (-86.68, -119.46, 31.98) mm, rotated rx -102.39 ry 0 rz -36.92 deg; joints [7.861, -86.559, 124.47, -159.785, 27.571, 151.373, -63.353]
  MoveL 1825 to (-86.92, -119.52, 31.09) mm, rotated rx -102.04 ry 0 rz -36.98 deg; joints [7.743, -86.595, 124.47, -160.001, 27.506, 151.88, -63.291]
  MoveL 1826 to (-87.44, -119.42, 30.02) mm, rotated rx -102.04 ry 0 rz -36.98 deg; joints [7.687, -86.585, 124.456, -160.125, 27.506, 151.978, -63.271]
  MoveL 1827 to (-88.11, -119.1, 29.31) mm, rotated rx -101.98 ry 0 rz -37.03 deg; joints [7.634, -86.564, 124.433, -160.243, 27.506, 152.137, -63.203]
  MoveL 1828 to (-90.45, -117.76, 27.55) mm, rotated rx -101.3 ry 0 rz -38.06 deg; joints [7.401, -86.631, 124.433, -160.676, 27.381, 153.143, -62.171]
  MoveL 1829 to (-90.79, -117.56, 27.27) mm, rotated rx -101.22 ry 0 rz -38.18 deg; joints [7.37, -86.636, 124.433, -160.741, 27.377, 153.274, -62.05]
  MoveL 1830 to (-93.09, -116.11, 25.68) mm, rotated rx -100.61 ry 0 rz -39.21 deg; joints [7.159, -86.693, 124.433, -161.138, 27.265, 154.188, -61.015]
  MoveL 1831 to (-95.54, -114.51, 23.8) mm, rotated rx -99.86 ry 0 rz -40.37 deg; joints [6.904, -86.762, 124.433, -161.615, 27.122, 155.298, -59.878]
  MoveL 1832 to (-96.15, -114.07, 23.47) mm, rotated rx -99.86 ry 0 rz -40.37 deg; joints [6.882, -86.714, 124.389, -161.664, 27.122, 155.338, -59.877]
  MoveL 1833 to (-96.7, -113.64, 23.29) mm, rotated rx -99.79 ry 0 rz -40.63 deg; joints [6.858, -86.72, 124.389, -161.709, 27.11, 155.441, -59.609]
  MoveL 1834 to (-100.85, -110.19, 22.17) mm, rotated rx -99.37 ry 0 rz -42.66 deg; joints [6.711, -86.751, 124.389, -161.998, 27.047, 156.085, -57.579]
  MoveL 1835 to (-102.57, -109.05, 19.9) mm, rotated rx -98.21 ry 0 rz -43.95 deg; joints [6.349, -86.888, 124.389, -162.608, 26.708, 157.697, -56.412]
  MoveL 1836 to (-103.23, -108.52, 19.3) mm, rotated rx -98.21 ry 0 rz -43.95 deg; joints [6.314, -86.837, 124.343, -162.688, 26.708, 157.762, -56.408]
  MoveL 1837 to (-103.63, -108.19, 19.07) mm, rotated rx -98.12 ry 0 rz -44.15 deg; joints [6.284, -86.844, 124.343, -162.747, 26.693, 157.894, -56.211]
  MoveL 1838 to (-108.47, -103.62, 17.48) mm, rotated rx -97.57 ry 0 rz -46.53 deg; joints [6.082, -86.868, 124.343, -163.172, 26.647, 158.783, -53.81]
  MoveL 1839 to (-110.72, -101.49, 15.76) mm, rotated rx -96.83 ry 0 rz -47.95 deg; joints [5.836, -86.941, 124.343, -163.621, 26.455, 159.87, -52.459]
  MoveL 1840 to (-111.18, -101.03, 15.52) mm, rotated rx -96.83 ry 0 rz -47.95 deg; joints [5.819, -86.897, 124.304, -163.658, 26.455, 159.9, -52.46]
  MoveL 1841 to (-111.55, -100.62, 15.43) mm, rotated rx -96.81 ry 0 rz -48.01 deg; joints [5.809, -86.871, 124.281, -163.681, 26.455, 159.933, -52.398]
  MoveL 1842 to (-112.64, -99.43, 15.33) mm, rotated rx -96.77 ry 0 rz -48.63 deg; joints [5.795, -86.874, 124.281, -163.708, 26.449, 159.994, -51.783]
  MoveL 1843 to (-114.5, -97.43, 14.34) mm, rotated rx -96.35 ry 0 rz -49.91 deg; joints [5.655, -86.925, 124.281, -163.949, 26.306, 160.599, -50.56]
  MoveL 1844 to (-114.93, -96.94, 14.2) mm, rotated rx -96.33 ry 0 rz -50.01 deg; joints [5.641, -86.9, 124.259, -163.979, 26.306, 160.642, -50.458]
  MoveL 1845 to (-116.59, -94.97, 13.94) mm, rotated rx -96.24 ry 0 rz -50.93 deg; joints [5.608, -86.897, 124.256, -164.055, 26.306, 160.792, -49.536]
  MoveL 1846 to (-116.84, -94.68, 13.79) mm, rotated rx -96.15 ry 0 rz -51.24 deg; joints [5.582, -86.919, 124.256, -164.079, 26.243, 160.893, -49.263]
  MoveL 1847 to (-120.24, -90.43, 12.79) mm, rotated rx -95.79 ry 0 rz -53.22 deg; joints [5.453, -86.93, 124.256, -164.356, 26.21, 161.474, -47.273]
  MoveL 1848 to (-136.18, -102.35, 14.8) mm, rotated rx -95.79 ry 0 rz -53.22 deg; joints [5.606, -87.891, 124.256, -164.247, 26.772, 161.29, -45.782]
  Set speed (1000.0 mm/s)
  MoveL 1849 to (-140.14, -95.07, 23.87) mm, rotated rx -98.56 ry 0 rz -55.2 deg; joints [6.664, -87.59, 124.256, -162.336, 27.563, 157.051, -43.542]
  Set speed (5.0 mm/s)
  MoveL 1850 to (-123.9, -83.78, 20.89) mm, rotated rx -98.56 ry 0 rz -55.2 deg; joints [6.456, -86.641, 124.256, -162.522, 26.97, 157.309, -45.036]
  Set speed (16.7 mm/s)
  MoveL 1851 to (-124.07, -83.45, 21.18) mm, rotated rx -98.78 ry 0 rz -55.45 deg; joints [6.519, -86.639, 124.257, -162.381, 26.97, 156.973, -44.805]
  MoveL 1852 to (-124.96, -81.65, 22.89) mm, rotated rx -99.43 ry 0 rz -56.21 deg; joints [6.745, -86.586, 124.257, -161.946, 27.085, 155.988, -44.033]
  MoveL 1853 to (-125.25, -80.96, 23.76) mm, rotated rx -99.82 ry 0 rz -56.25 deg; joints [6.872, -86.529, 124.257, -161.749, 27.223, 155.453, -43.937]
  MoveL 1854 to (-124.73, -80.95, 26.31) mm, rotated rx -100.71 ry 0 rz -56.35 deg; joints [7.191, -86.467, 124.257, -161.107, 27.328, 154.066, -43.878]
  MoveL 1855 to (-125.37, -79.47, 27.83) mm, rotated rx -101.3 ry 0 rz -56.96 deg; joints [7.392, -86.412, 124.257, -160.731, 27.435, 153.197, -43.264]
  MoveL 1856 to (-125.5, -79.1, 28.27) mm, rotated rx -101.37 ry 0 rz -57.01 deg; joints [7.429, -86.392, 124.257, -160.678, 27.482, 153.086, -43.186]
  MoveL 1857 to (-125.87, -77.67, 30.51) mm, rotated rx -102.15 ry 0 rz -57.5 deg; joints [7.706, -86.305, 124.257, -160.179, 27.651, 151.936, -42.689]
  MoveL 1858 to (-126.01, -77.35, 30.76) mm, rotated rx -102.41 ry 0 rz -57.76 deg; joints [7.775, -86.299, 124.259, -160.026, 27.651, 151.551, -42.452]
  MoveL 1859 to (-128.01, -71.29, 36.59) mm, rotated rx -104.7 ry 0 rz -60.21 deg; joints [8.548, -86.045, 124.259, -158.628, 28.079, 148.222, -40.033]
  MoveL 1860 to (-128.08, -70.51, 37.83) mm, rotated rx -104.7 ry 0 rz -60.21 deg; joints [8.607, -85.994, 124.259, -158.58, 28.197, 148.2, -39.976]
  MoveL 1861 to (-127.99, -70.35, 38.41) mm, rotated rx -104.8 ry 0 rz -60.23 deg; joints [8.655, -85.975, 124.259, -158.5, 28.231, 148.05, -39.954]
  MoveL 1862 to (-127.73, -70.1, 39.72) mm, rotated rx -105.31 ry 0 rz -60.26 deg; joints [8.827, -85.912, 124.259, -158.198, 28.331, 147.316, -39.929]
  MoveL 1863 to (-127.97, -68.59, 41.54) mm, rotated rx -106.53 ry 0 rz -61.02 deg; joints [9.171, -85.799, 124.259, -157.561, 28.477, 145.625, -39.236]
  MoveL 1864 to (-128.66, -66.29, 43.13) mm, rotated rx -107.37 ry 0 rz -62.17 deg; joints [9.423, -85.72, 124.259, -157.081, 28.562, 144.432, -38.15]
  MoveL 1865 to (-128.78, -65.7, 43.67) mm, rotated rx -107.37 ry 0 rz -62.17 deg; joints [9.447, -85.678, 124.243, -157.07, 28.615, 144.432, -38.126]
  MoveL 1866 to (-128.8, -65.27, 44.25) mm, rotated rx -107.44 ry 0 rz -62.22 deg; joints [9.489, -85.65, 124.243, -157.018, 28.671, 144.33, -38.054]
  MoveL 1867 to (-128.69, -64.21, 46.08) mm, rotated rx -108.17 ry 0 rz -62.58 deg; joints [9.728, -85.548, 124.243, -156.615, 28.817, 143.317, -37.725]
  MoveL 1868 to (-128.72, -63.87, 46.47) mm, rotated rx -108.46 ry 0 rz -62.79 deg; joints [9.808, -85.522, 124.243, -156.464, 28.841, 142.913, -37.539]
  MoveL 1869 to (-129.16, -61.26, 48.69) mm, rotated rx -109.5 ry 0 rz -63.93 deg; joints [10.128, -85.391, 124.243, -155.903, 29, 141.475, -36.459]
  MoveL 1870 to (-129.09, -61.41, 48.69) mm, rotated rx -108.26 ry 0 rz -65.38 deg; joints [9.889, -85.659, 124.243, -155.964, 28.405, 142.663, -35.305]
  MoveL 1871 to (-128.97, -64.41, 44.99) mm, rotated rx -106.78 ry 0 rz -64.27 deg; joints [9.404, -85.867, 124.243, -156.792, 28.109, 144.731, -36.363]
  MoveL 1872 to (-128.99, -64.74, 44.48) mm, rotated rx -106.78 ry 0 rz -64.27 deg; joints [9.38, -85.889, 124.243, -156.809, 28.06, 144.736, -36.386]
  MoveL 1873 to (-129.25, -65.47, 42.6) mm, rotated rx -106.16 ry 0 rz -64.1 deg; joints [9.159, -85.982, 124.243, -157.184, 27.916, 145.626, -36.549]
  MoveL 1874 to (-129.24, -65.64, 42.38) mm, rotated rx -105.8 ry 0 rz -63.91 deg; joints [9.073, -86.003, 124.243, -157.361, 27.9, 146.121, -36.702]
  MoveL 1875 to (-128.22, -70.09, 38.13) mm, rotated rx -103.96 ry 0 rz -62.03 deg; joints [8.477, -86.208, 124.243, -158.45, 27.594, 148.766, -38.517]
  MoveL 1876 to (-128.17, -70.82, 36.94) mm, rotated rx -103.96 ry 0 rz -62.03 deg; joints [8.419, -86.256, 124.243, -158.498, 27.483, 148.789, -38.57]
  MoveL 1877 to (-128.22, -70.97, 36.46) mm, rotated rx -103.77 ry 0 rz -61.99 deg; joints [8.355, -86.278, 124.243, -158.614, 27.446, 149.064, -38.61]
  MoveL 1878 to (-128.78, -71.68, 32.9) mm, rotated rx -101.85 ry 0 rz -61.51 deg; joints [7.769, -86.43, 124.243, -159.76, 27.222, 151.859, -39.006]
  MoveL 1879 to (-127.36, -75.53, 29.71) mm, rotated rx -100.61 ry 0 rz -59.93 deg; joints [7.345, -86.553, 124.243, -160.554, 26.993, 153.699, -40.579]
  MoveL 1880 to (-127.19, -76.01, 29.19) mm, rotated rx -100.61 ry 0 rz -59.93 deg; joints [7.321, -86.581, 124.244, -160.564, 26.924, 153.699, -40.619]
  MoveL 1881 to (-127.12, -76.28, 28.8) mm, rotated rx -100.45 ry 0 rz -59.83 deg; joints [7.268, -86.595, 124.244, -160.664, 26.896, 153.928, -40.727]
  MoveL 1882 to (-127.06, -76.58, 28.26) mm, rotated rx -100.45 ry 0 rz -59.83 deg; joints [7.242, -86.614, 124.244, -160.692, 26.848, 153.945, -40.751]
  MoveL 1883 to (-126.91, -77.99, 24.86) mm, rotated rx -99.14 ry 0 rz -59.33 deg; joints [6.79, -86.73, 124.244, -161.561, 26.613, 155.922, -41.259]
  MoveL 1884 to (-124.48, -82.65, 21.91) mm, rotated rx -97.52 ry 0 rz -56.89 deg; joints [6.288, -86.799, 124.244, -162.621, 26.493, 158.381, -43.63]
  MoveL 1885 to (-124.18, -83.21, 21.54) mm, rotated rx -97.39 ry 0 rz -56.67 deg; joints [6.241, -86.812, 124.244, -162.709, 26.462, 158.579, -43.855]
  MoveL 1886 to (-140.53, -94.5, 23.78) mm, rotated rx -97.34 ry 0 rz -56.62 deg; joints [6.403, -87.78, 124.244, -162.594, 27.005, 158.419, -42.435]
  Set speed (1000.0 mm/s)
  MoveL 1887 to (-136.26, -102.31, 14.35) mm, rotated rx -94.11 ry 0 rz -53.56 deg; joints [5.215, -87.982, 124.244, -164.97, 26.466, 163.533, -45.571]
  Set speed (5.0 mm/s)
  MoveL 1888 to (-120.21, -90.46, 12.91) mm, rotated rx -94.11 ry 0 rz -53.56 deg; joints [5.112, -87.173, 124.545, -165.254, 26.466, 163.895, -46.648]
  Set speed (16.7 mm/s)
  MoveL 1889 to (-119.01, -92.24, 11.51) mm, rotated rx -93.58 ry 0 rz -52.75 deg; joints [4.924, -87.199, 124.546, -165.638, 26.384, 164.732, -47.482]
  MoveL 1890 to (-118.99, -92.27, 11.51) mm, rotated rx -93.45 ry 0 rz -51.97 deg; joints [4.885, -87.059, 124.423, -165.726, 26.384, 164.931, -48.267]
  MoveL 1891 to (-117.48, -94.12, 12.12) mm, rotated rx -93.68 ry 0 rz -51.06 deg; joints [4.967, -87.049, 124.423, -165.559, 26.42, 164.567, -49.162]
  MoveL 1892 to (-117.07, -94.62, 12.21) mm, rotated rx -93.69 ry 0 rz -50.98 deg; joints [4.975, -87.079, 124.449, -165.541, 26.42, 164.545, -49.243]
  MoveL 1893 to (-115.83, -96.13, 12.2) mm, rotated rx -93.68 ry 0 rz -50.32 deg; joints [4.975, -87.095, 124.463, -165.541, 26.418, 164.551, -49.905]
  MoveL 1894 to (-114.39, -97.74, 13.03) mm, rotated rx -94.06 ry 0 rz -49.17 deg; joints [5.096, -87.043, 124.463, -165.344, 26.576, 164.034, -50.973]
  MoveL 1895 to (-113.7, -98.51, 13.23) mm, rotated rx -94.09 ry 0 rz -48.96 deg; joints [5.116, -87.074, 124.491, -165.3, 26.576, 163.967, -51.184]
  MoveL 1896 to (-109.74, -102.86, 13.59) mm, rotated rx -94.22 ry 0 rz -46.8 deg; joints [5.163, -87.077, 124.493, -165.194, 26.576, 163.753, -53.351]
  MoveL 1897 to (-109.47, -103.13, 13.67) mm, rotated rx -94.25 ry 0 rz -46.56 deg; joints [5.175, -87.066, 124.493, -165.185, 26.61, 163.71, -53.57]
  MoveL 1898 to (-106.27, -106.28, 14.78) mm, rotated rx -94.69 ry 0 rz -44.77 deg; joints [5.327, -87.034, 124.493, -164.891, 26.703, 163.041, -55.33]
  MoveL 1899 to (-105.7, -106.84, 14.84) mm, rotated rx -94.69 ry 0 rz -44.77 deg; joints [5.335, -87.092, 124.544, -164.872, 26.703, 163.025, -55.325]
  MoveL 1900 to (-104.6, -108.02, 14.08) mm, rotated rx -94.69 ry 0 rz -44.77 deg; joints [5.303, -87.188, 124.594, -164.885, 26.586, 163.025, -55.392]
  MoveL 1901 to (-104.3, -108.37, 13.6) mm, rotated rx -94.51 ry 0 rz -44.59 deg; joints [5.239, -87.198, 124.594, -165.015, 26.558, 163.309, -55.572]
  MoveL 1902 to (-103.93, -108.96, 11.62) mm, rotated rx -94.51 ry 0 rz -44.59 deg; joints [5.14, -87.24, 124.594, -165.175, 26.433, 163.428, -55.637]
  MoveL 1903 to (-104.45, -108.84, 7.2) mm, rotated rx -92.83 ry 0 rz -44.77 deg; joints [4.546, -87.316, 124.594, -166.393, 26.179, 166.072, -55.53]
  MoveL 1904 to (-104.58, -108.76, 6.57) mm, rotated rx -92.77 ry 0 rz -44.78 deg; joints [4.5, -87.317, 124.594, -166.493, 26.171, 166.214, -55.509]
  MoveL 1905 to (-104.79, -108.62, 5.38) mm, rotated rx -92.25 ry 0 rz -44.9 deg; joints [4.325, -87.337, 124.594, -166.856, 26.093, 167.027, -55.421]
  MoveL 1906 to (-105.18, -108.3, 4.15) mm, rotated rx -91.97 ry 0 rz -45.03 deg; joints [4.201, -87.342, 124.594, -167.124, 26.062, 167.519, -55.297]
  MoveL 1907 to (-108.36, -105.17, -2.01) mm, rotated rx -89.8 ry 0 rz -46.62 deg; joints [3.408, -87.385, 124.594, -168.816, 25.789, 171.045, -53.802]
  MoveL 1908 to (-108.65, -104.83, -3.64) mm, rotated rx -88.89 ry 0 rz -46.93 deg; joints [3.125, -87.41, 124.594, -169.407, 25.643, 172.425, -53.573]
  MoveL 1909 to (-108.84, -104.61, -4.29) mm, rotated rx -88.89 ry 0 rz -46.93 deg; joints [3.091, -87.392, 124.581, -169.485, 25.643, 172.488, -53.573]
  MoveL 1910 to (-109.13, -104.27, -4.96) mm, rotated rx -88.64 ry 0 rz -47.1 deg; joints [3.001, -87.394, 124.581, -169.681, 25.61, 172.902, -53.423]
  MoveL 1911 to (-113.05, -99.53, -11.02) mm, rotated rx -86.5 ry 0 rz -49.3 deg; joints [2.22, -87.395, 124.609, -171.418, 25.448, 176.449, -51.309]
  MoveL 1912 to (-113.34, -99.15, -11.43) mm, rotated rx -86.38 ry 0 rz -49.44 deg; joints [2.173, -87.389, 124.61, -171.526, 25.448, 176.654, -51.172]
  MoveL 1913 to (-115.31, -96.51, -13.99) mm, rotated rx -85.43 ry 0 rz -50.66 deg; joints [1.835, -87.389, 124.64, -172.293, 25.411, 178.225, -49.983]
  MoveL 1914 to (-115.68, -96.01, -14.39) mm, rotated rx -85.34 ry 0 rz -50.81 deg; joints [1.794, -87.373, 124.63, -172.387, 25.411, 178.392, -49.837]
  MoveL 1915 to (-118.09, -92.7, -16.37) mm, rotated rx -84.63 ry 0 rz -52.28 deg; joints [1.538, -87.363, 124.656, -172.975, 25.41, 179.583, -48.369]
  MoveL 1916 to (-118.46, -92.16, -16.77) mm, rotated rx -84.44 ry 0 rz -52.61 deg; joints [1.474, -87.367, 124.656, -173.11, 25.368, 179.886, -48.075]
  MoveL 1917 to (-121.85, -86.42, -22.18) mm, rotated rx -82.29 ry 0 rz -55.26 deg; joints [0.73, -87.367, 124.759, -174.811, 25.327, 183.419, -45.504]
  MoveL 1918 to (-122.46, -84.98, -24.25) mm, rotated rx -81.33 ry 0 rz -56.01 deg; joints [0.415, -87.368, 124.798, -175.525, 25.276, 184.957, -44.828]
  MoveL 1919 to (-122.65, -84.59, -24.68) mm, rotated rx -81.33 ry 0 rz -56.01 deg; joints [0.393, -87.334, 124.773, -175.577, 25.276, 185, -44.834]
  MoveL 1920 to (-122.81, -84.27, -24.97) mm, rotated rx -81.22 ry 0 rz -56.15 deg; joints [0.354, -87.332, 124.778, -175.665, 25.276, 185.183, -44.7]
  MoveL 1921 to (-124.4, -81.2, -27.15) mm, rotated rx -80.44 ry 0 rz -57.38 deg; joints [0.074, -87.293, 124.797, -176.309, 25.276, 186.484, -43.504]
  MoveL 1922 to (-124.78, -79.6, -30.03) mm, rotated rx -78.99 ry 0 rz -58.31 deg; joints [-0.388, -87.293, 124.874, -177.363, 25.222, 188.796, -42.69]
  MoveL 1923 to (-124.89, -79.17, -30.67) mm, rotated rx -78.81 ry 0 rz -58.43 deg; joints [-0.46, -87.276, 124.874, -177.526, 25.222, 189.106, -42.582]
  MoveL 1924 to (-125.14, -77.59, -33.5) mm, rotated rx -77.62 ry 0 rz -59.06 deg; joints [-0.861, -87.23, 124.923, -178.447, 25.222, 191.048, -42.034]
  MoveL 1925 to (-125.14, -77.57, -33.6) mm, rotated rx -76.62 ry 0 rz -59.02 deg; joints [-1.082, -87.185, 124.934, -178.953, 25.222, 192.457, -42.132]
  MoveL 1926 to (-124.65, -77.98, -34.49) mm, rotated rx -76.27 ry 0 rz -58.78 deg; joints [-1.201, -87.164, 124.944, -179.226, 25.222, 193.023, -42.397]
  MoveL 1927 to (-124.35, -78.16, -35.13) mm, rotated rx -76.27 ry 0 rz -58.78 deg; joints [-1.233, -87.181, 124.968, -179.3, 25.222, 193.083, -42.403]
  MoveL 1928 to (-124.19, -78.22, -35.56) mm, rotated rx -76.11 ry 0 rz -58.73 deg; joints [-1.291, -87.171, 124.972, -179.432, 25.222, 193.358, -42.47]
  MoveL 1929 to (-123.95, -78.19, -36.45) mm, rotated rx -76.11 ry 0 rz -58.73 deg; joints [-1.336, -87.17, 124.983, -179.536, 25.222, 193.443, -42.481]
  MoveL 1930 to (-123.38, -77.54, -39.6) mm, rotated rx -74.87 ry 0 rz -58.83 deg; joints [-1.76, -87.083, 125.016, -180.506, 25.222, 195.462, -42.5]
  MoveL 1931 to (-120.74, -79.41, -43.84) mm, rotated rx -72.6 ry 0 rz -57.5 deg; joints [-2.455, -86.882, 125.035, -182.095, 25.222, 199.014, -44.067]
  MoveL 1932 to (-120.21, -79.55, -45.03) mm, rotated rx -72.6 ry 0 rz -57.5 deg; joints [-2.516, -86.897, 125.065, -182.233, 25.222, 199.125, -44.085]
  MoveL 1933 to (-119.97, -79.45, -45.84) mm, rotated rx -72.28 ry 0 rz -57.48 deg; joints [-2.624, -86.866, 125.071, -182.482, 25.222, 199.647, -44.142]
  MoveL 1934 to (-117.99, -78.14, -52.73) mm, rotated rx -69.57 ry 0 rz -57.5 deg; joints [-3.536, -86.579, 125.115, -184.56, 25.222, 204.023, -44.501]
  MoveL 1935 to (-116.68, -77.5, -56.45) mm, rotated rx -68.02 ry 0 rz -57.43 deg; joints [-4.038, -86.394, 125.134, -185.704, 25.222, 206.477, -44.807]
  MoveL 1936 to (-116.44, -76.93, -57.7) mm, rotated rx -68.02 ry 0 rz -57.43 deg; joints [-4.101, -86.353, 125.134, -185.839, 25.262, 206.582, -44.812]
  MoveL 1937 to (-116.45, -76.65, -58.07) mm, rotated rx -67.87 ry 0 rz -57.53 deg; joints [-4.15, -86.334, 125.135, -185.951, 25.262, 206.822, -44.739]
  MoveL 1938 to (-116.52, -76.14, -58.6) mm, rotated rx -67.87 ry 0 rz -57.53 deg; joints [-4.176, -86.294, 125.118, -186.005, 25.286, 206.864, -44.739]
  MoveL 1939 to (-117.45, -71.82, -62.09) mm, rotated rx -66.42 ry 0 rz -59.26 deg; joints [-4.641, -86.102, 125.132, -187.061, 25.286, 209.144, -43.256]
  MoveL 1940 to (-117.61, -71.24, -62.45) mm, rotated rx -66.42 ry 0 rz -59.26 deg; joints [-4.659, -86.069, 125.132, -187.084, 25.359, 209.158, -43.217]
  MoveL 1941 to (-117.78, -70.77, -62.67) mm, rotated rx -66.33 ry 0 rz -59.46 deg; joints [-4.688, -86.056, 125.133, -187.149, 25.358, 209.3, -43.032]
  MoveL 1942 to (-119.62, -65.95, -64.4) mm, rotated rx -65.65 ry 0 rz -61.49 deg; joints [-4.911, -85.944, 125.133, -187.648, 25.377, 210.379, -41.112]
  MoveL 1943 to (-119.93, -63.2, -66.55) mm, rotated rx -64.56 ry 0 rz -62.91 deg; joints [-5.235, -85.854, 125.192, -188.381, 25.377, 212.041, -39.875]
  MoveL 1944 to (-120.07, -62.36, -67.09) mm, rotated rx -64.4 ry 0 rz -63.16 deg; joints [-5.292, -85.816, 125.192, -188.502, 25.404, 212.29, -39.644]
  MoveL 1945 to (-120.27, -59.5, -69.25) mm, rotated rx -63.41 ry 0 rz -64.4 deg; joints [-5.595, -85.684, 125.214, -189.185, 25.404, 213.819, -38.601]
  MoveL 1946 to (-120.29, -59.56, -69.2) mm, rotated rx -62.39 ry 0 rz -64.66 deg; joints [-5.791, -85.636, 125.26, -189.626, 25.404, 215.176, -38.458]
  MoveL 1947 to (-119.61, -59.72, -70.24) mm, rotated rx -61.95 ry 0 rz -64.47 deg; joints [-5.926, -85.565, 125.263, -189.931, 25.404, 215.852, -38.734]
  MoveL 1948 to (-119.15, -59.77, -70.98) mm, rotated rx -61.71 ry 0 rz -64.39 deg; joints [-6.01, -85.525, 125.268, -190.12, 25.404, 216.244, -38.869]
  MoveL 1949 to (-118.82, -59.72, -71.58) mm, rotated rx -61.71 ry 0 rz -64.39 deg; joints [-6.04, -85.515, 125.275, -190.188, 25.404, 216.297, -38.889]
  MoveL 1950 to (-115.87, -58.28, -77.36) mm, rotated rx -59.18 ry 0 rz -64.4 deg; joints [-6.799, -85.084, 125.288, -191.893, 25.404, 220.127, -39.434]
  MoveL 1951 to (-115.4, -57.54, -78.6) mm, rotated rx -59.18 ry 0 rz -64.4 deg; joints [-6.86, -85.027, 125.288, -192.005, 25.461, 220.207, -39.442]
  MoveL 1952 to (-115.3, -56.99, -79.15) mm, rotated rx -58.94 ry 0 rz -64.61 deg; joints [-6.932, -84.983, 125.29, -192.167, 25.461, 220.575, -39.296]
  MoveL 1953 to (-115.31, -56.09, -79.78) mm, rotated rx -58.94 ry 0 rz -64.61 deg; joints [-6.962, -84.928, 125.29, -192.19, 25.565, 220.584, -39.25]
  MoveL 1954 to (-116.04, -50.67, -82.28) mm, rotated rx -57.81 ry 0 rz -66.97 deg; joints [-7.291, -84.722, 125.298, -192.924, 25.565, 222.268, -37.157]
  MoveL 1955 to (-115.37, -50.42, -83.39) mm, rotated rx -56.63 ry 0 rz -67.52 deg; joints [-7.564, -84.641, 125.383, -193.532, 25.565, 223.908, -36.818]
  MoveL 1956 to (-115.05, -50.09, -84.03) mm, rotated rx -56.53 ry 0 rz -67.54 deg; joints [-7.613, -84.602, 125.383, -193.634, 25.58, 224.084, -36.832]
  MoveL 1957 to (-113.62, -47.98, -87.15) mm, rotated rx -55.08 ry 0 rz -68.2 deg; joints [-8.021, -84.326, 125.396, -194.537, 25.58, 226.199, -36.534]
  MoveL 1958 to (-113.36, -47.37, -87.82) mm, rotated rx -54.96 ry 0 rz -68.3 deg; joints [-8.075, -84.276, 125.396, -194.643, 25.609, 226.399, -36.465]
  MoveL 1959 to (-113.25, -46.78, -88.28) mm, rotated rx -54.96 ry 0 rz -68.3 deg; joints [-8.097, -84.237, 125.396, -194.658, 25.674, 226.403, -36.442]
  MoveL 1960 to (-113, -43.69, -90.16) mm, rotated rx -54.07 ry 0 rz -69.62 deg; joints [-8.342, -84.063, 125.406, -195.198, 25.674, 227.687, -35.35]
  MoveL 1961 to (-111.7, -40.57, -93.19) mm, rotated rx -52.42 ry 0 rz -71.04 deg; joints [-8.772, -83.783, 125.456, -196.144, 25.674, 230.028, -34.343]
  MoveL 1962 to (-111.45, -39.65, -93.88) mm, rotated rx -52.22 ry 0 rz -71.29 deg; joints [-8.839, -83.717, 125.456, -196.275, 25.703, 230.322, -34.144]
  MoveL 1963 to (-110.29, -33.42, -97.61) mm, rotated rx -50.45 ry 0 rz -73.95 deg; joints [-9.311, -83.335, 125.474, -197.303, 25.703, 232.826, -31.978]
  MoveL 1964 to (-110.16, -32.55, -98.04) mm, rotated rx -50.3 ry 0 rz -74.24 deg; joints [-9.356, -83.286, 125.474, -197.389, 25.725, 233.037, -31.723]
  MoveL 1965 to (-110.14, -31.93, -98.28) mm, rotated rx -50.3 ry 0 rz -74.24 deg; joints [-9.364, -83.236, 125.446, -197.394, 25.743, 233.037, -31.727]
  MoveL 1966 to (-110.3, -24.54, -100.19) mm, rotated rx -49.33 ry 0 rz -77.88 deg; joints [-9.612, -83.035, 125.466, -197.932, 25.743, 234.383, -28.366]
  MoveL 1967 to (-110.37, -23.8, -100.3) mm, rotated rx -49.33 ry 0 rz -77.88 deg; joints [-9.612, -82.976, 125.42, -197.93, 25.743, 234.38, -28.379]
  MoveL 1968 to (-110.46, -23.32, -100.31) mm, rotated rx -49.33 ry 0 rz -78.12 deg; joints [-9.613, -82.975, 125.42, -197.934, 25.743, 234.389, -28.132]
  MoveL 1969 to (-111.37, -19.04, -100.2) mm, rotated rx -49.38 ry 0 rz -80.26 deg; joints [-9.598, -82.973, 125.408, -197.9, 25.743, 234.31, -25.986]
  MoveL 1970 to (-111.19, -17.5, -100.68) mm, rotated rx -49.07 ry 0 rz -81.53 deg; joints [-9.679, -82.988, 125.479, -198.077, 25.743, 234.751, -24.782]
  MoveL 1971 to (-111.18, -16.84, -100.81) mm, rotated rx -49.07 ry 0 rz -81.53 deg; joints [-9.68, -82.935, 125.439, -198.079, 25.743, 234.751, -24.795]
  MoveL 1972 to (-111.39, -15.31, -100.82) mm, rotated rx -49.07 ry 0 rz -82.16 deg; joints [-9.679, -82.91, 125.418, -198.075, 25.743, 234.749, -24.177]
  MoveL 1973 to (-111.16, -13.52, -101.33) mm, rotated rx -48.75 ry 0 rz -83.5 deg; joints [-9.76, -82.913, 125.481, -198.253, 25.743, 235.194, -22.914]
  MoveL 1974 to (-111.2, -12.35, -101.43) mm, rotated rx -48.75 ry 0 rz -83.5 deg; joints [-9.756, -82.822, 125.408, -198.242, 25.743, 235.184, -22.93]
  MoveL 1975 to (-111.31, -11.84, -101.38) mm, rotated rx -48.77 ry 0 rz -83.77 deg; joints [-9.75, -82.828, 125.407, -198.228, 25.743, 235.148, -22.653]
  MoveL 1976 to (-112.07, -10.29, -100.7) mm, rotated rx -48.77 ry 0 rz -83.77 deg; joints [-9.706, -82.736, 125.302, -198.13, 25.743, 235.074, -22.631]
  MoveL 1977 to (-115.12, -7.08, -97.49) mm, rotated rx -50.4 ry 0 rz -85.53 deg; joints [-9.291, -83.077, 125.269, -197.232, 25.743, 232.817, -20.406]
  MoveL 1978 to (-116.27, -6.59, -96.15) mm, rotated rx -50.4 ry 0 rz -85.53 deg; joints [-9.222, -83.087, 125.228, -197.082, 25.743, 232.708, -20.341]
  MoveL 1979 to (-116.81, -6.76, -95.49) mm, rotated rx -50.49 ry 0 rz -85.52 deg; joints [-9.175, -83.131, 125.228, -196.984, 25.735, 232.545, -20.302]
  MoveL 1980 to (-117.52, -7.19, -94.57) mm, rotated rx -50.93 ry 0 rz -85.34 deg; joints [-9.059, -83.223, 125.22, -196.731, 25.735, 231.921, -20.36]
  MoveL 1981 to (-117.57, -7.2, -94.5) mm, rotated rx -51.73 ry 0 rz -85.44 deg; joints [-8.926, -83.341, 125.22, -196.447, 25.724, 230.925, -20.127]
  MoveL 1982 to (-119.21, -5.88, -92.53) mm, rotated rx -52.69 ry 0 rz -86.14 deg; joints [-8.67, -83.537, 125.207, -195.889, 25.724, 229.562, -19.167]
  MoveL 1983 to (-119.61, -5.59, -92.04) mm, rotated rx -52.87 ry 0 rz -86.25 deg; joints [-8.616, -83.572, 125.199, -195.769, 25.724, 229.294, -19.001]
  MoveL 1984 to (-122.12, -3.99, -88.75) mm, rotated rx -54.38 ry 0 rz -87.05 deg; joints [-8.199, -83.872, 125.177, -194.855, 25.724, 227.116, -17.799]
  MoveL 1985 to (-123.65, -1.68, -86.68) mm, rotated rx -55.61 ry 0 rz -88.37 deg; joints [-7.884, -84.12, 125.177, -194.18, 25.686, 225.385, -16.212]
  MoveL 1986 to (-124.31, -0.98, -85.75) mm, rotated rx -55.86 ry 0 rz -88.54 deg; joints [-7.793, -84.156, 125.152, -193.978, 25.686, 224.984, -15.964]
